LIN {X 0,Y 542.903,Z 219.007,A -85,B 0,C 180,E1 24562.487,E2 24562.487} C_VEL
LIN {X 0,Y 541.878,Z 217.291,A -85,B 0,C 180,E1 24561.084,E2 24561.084} C_VEL
LIN {X 0,Y 539.286,Z 215.915,A -85,B 0,C 180,E1 24558.559,E2 24558.559} C_VEL
LIN {X 0,Y 536.919,Z 213.82,A -85,B 0,C 180,E1 24556.541,E2 24556.541} C_VEL
LIN {X 0,Y 534.543,Z 210.096,A -85,B 0,C 180,E1 24554.71,E2 24554.71} C_VEL
LIN {X 0,Y 531.153,Z 208.109,A -85,B 0,C 180,E1 24552.586,E2 24552.586} C_VEL
LIN {X 0,Y 528.889,Z 205.137,A -85,B 0,C 180,E1 24551.198,E2 24551.198} C_VEL
LIN {X 0,Y 527.514,Z 203.01,A -85,B 0,C 180,E1 24550.4,E2 24550.4} C_VEL
LIN {X 0,Y 524.38,Z 201.255,A -85,B 0,C 180,E1 24548.817,E2 24548.817} C_VEL
LIN {X 0,Y 522.406,Z 198.666,A -85,B 0,C 180,E1 24547.792,E2 24547.792} C_VEL
LIN {X 0,Y 521.741,Z 196.733,A -85,B 0,C 180,E1 24547.193,E2 24547.193} C_VEL
LIN {X 0,Y 521.717,Z 196.18,A -85,B 0,C 180,E1 24546.271,E2 24546.271} C_VEL
LIN {X 0,Y 521.67,Z 196.188,A -85,B 0,C 180,E1 24542.863,E2 24542.863} C_VEL
LIN {X 0,Y 521.655,Z 196.188,A -85,B 0,C 180,E1 24539.478,E2 24539.478} C_VEL
LIN {X 0,Y 521.706,Z 196.182,A -85,B 0,C 180,E1 24536.239,E2 24536.239} C_VEL
LIN {X 0,Y 521.677,Z 196.188,A -85,B 0,C 180,E1 24532.867,E2 24532.867} C_VEL
LIN {X 0,Y 521.656,Z 196.187,A -85,B 0,C 180,E1 24529.549,E2 24529.549} C_VEL
LIN {X 0,Y 521.694,Z 196.184,A -85,B 0,C 180,E1 24526.227,E2 24526.227} C_VEL
LIN {X 0,Y 521.689,Z 196.187,A -85,B 0,C 180,E1 24522.876,E2 24522.876} C_VEL
LIN {X 0,Y 521.655,Z 196.188,A -85,B 0,C 180,E1 24519.607,E2 24519.607} C_VEL
LIN {X 0,Y 521.686,Z 196.144,A -85,B 0,C 180,E1 24516.317,E2 24516.317} C_VEL
LIN {X 0,Y 521.69,Z 196.17,A -85,B 0,C 180,E1 24512.926,E2 24512.926} C_VEL
LIN {X 0,Y 521.65,Z 196.155,A -85,B 0,C 180,E1 24509.639,E2 24509.639} C_VEL
LIN {X 0,Y 521.686,Z 196.134,A -85,B 0,C 180,E1 24506.402,E2 24506.402} C_VEL
LIN {X 0,Y 521.687,Z 196.186,A -85,B 0,C 180,E1 24503.094,E2 24503.094} C_VEL
LIN {X 0,Y 521.654,Z 196.185,A -85,B 0,C 180,E1 24499.779,E2 24499.779} C_VEL
LIN {X 0,Y 521.685,Z 196.169,A -85,B 0,C 180,E1 24496.479,E2 24496.479} C_VEL
LIN {X 0,Y 521.684,Z 196.173,A -85,B 0,C 180,E1 24493.213,E2 24493.213} C_VEL
LIN {X 0,Y 521.654,Z 196.185,A -85,B 0,C 180,E1 24489.822,E2 24489.822} C_VEL
LIN {X 0,Y 521.666,Z 196.176,A -85,B 0,C 180,E1 24486.383,E2 24486.383} C_VEL
LIN {X 0,Y 521.707,Z 196.167,A -85,B 0,C 180,E1 24483.076,E2 24483.076} C_VEL
LIN {X 0,Y 521.657,Z 196.185,A -85,B 0,C 180,E1 24479.78,E2 24479.78} C_VEL
LIN {X 0,Y 521.655,Z 196.174,A -85,B 0,C 180,E1 24476.263,E2 24476.263} C_VEL
LIN {X 0,Y 521.708,Z 196.163,A -85,B 0,C 180,E1 24472.954,E2 24472.954} C_VEL
LIN {X 0,Y 521.673,Z 196.183,A -85,B 0,C 180,E1 24469.62,E2 24469.62} C_VEL
LIN {X 0,Y 521.653,Z 196.179,A -85,B 0,C 180,E1 24466.25,E2 24466.25} C_VEL
LIN {X 0,Y 521.701,Z 196.166,A -85,B 0,C 180,E1 24462.989,E2 24462.989} C_VEL
LIN {X 0,Y 521.677,Z 196.186,A -85,B 0,C 180,E1 24459.701,E2 24459.701} C_VEL
LIN {X 0,Y 521.656,Z 196.185,A -85,B 0,C 180,E1 24456.36,E2 24456.36} C_VEL
LIN {X 0,Y 521.69,Z 196.137,A -85,B 0,C 180,E1 24453.013,E2 24453.013} C_VEL
LIN {X 0,Y 521.674,Z 196.16,A -85,B 0,C 180,E1 24449.804,E2 24449.804} C_VEL
LIN {X 0,Y 521.654,Z 196.173,A -85,B 0,C 180,E1 24446.479,E2 24446.479} C_VEL
LIN {X 0,Y 521.693,Z 196.178,A -85,B 0,C 180,E1 24443.137,E2 24443.137} C_VEL
LIN {X 0,Y 521.678,Z 196.156,A -85,B 0,C 180,E1 24439.876,E2 24439.876} C_VEL
LIN {X 0,Y 521.655,Z 196.17,A -85,B 0,C 180,E1 24436.518,E2 24436.518} C_VEL
LIN {X 0,Y 521.685,Z 196.174,A -85,B 0,C 180,E1 24433.169,E2 24433.169} C_VEL
LIN {X 0,Y 521.758,Z 196.445,A -85,B 0,C 180,E1 24431.589,E2 24431.589} C_VEL
LIN {X 0,Y 528.289,Z 215.738,A -85,B 0,C 180,E1 24428.585,E2 24428.585} C_VEL
LIN {X 0,Y 529.766,Z 220.377,A -85,B 0,C 180,E1 24427.913,E2 24427.913} C_VEL
LIN {X 0,Y 541.007,Z 241.596,A -85,B 0,C 180,E1 24426.622,E2 24426.622} C_VEL
LIN {X 0,Y 548.011,Z 256.158,A -85,B 0,C 180,E1 24425.852,E2 24425.852} C_VEL
LIN {X 0,Y 550.912,Z 271.289,A -85,B 0,C 180,E1 24425.399,E2 24425.399} C_VEL
LIN {X 0,Y 544.997,Z 522.592,A -85,B 0,C 180,E1 24421.909,E2 24421.909} C_VEL
LIN {X 0,Y 544.141,Z 540.067,A -85,B 0,C 180,E1 24421.568,E2 24421.568} C_VEL
LIN {X 0,Y 543,Z 557.267,A -85,B 0,C 180,E1 24421.118,E2 24421.118} C_VEL
LIN {X 0,Y 541.545,Z 575.435,A -85,B 0,C 180,E1 24420.509,E2 24420.509} C_VEL
LIN {X 0,Y 539.48,Z 597.06,A -85,B 0,C 180,E1 24419.595,E2 24419.595} C_VEL
LIN {X 0,Y 537.434,Z 615.482,A -85,B 0,C 180,E1 24418.621,E2 24418.621} C_VEL
LIN {X 0,Y 535.499,Z 631.43,A -85,B 0,C 180,E1 24417.63,E2 24417.63} C_VEL
LIN {X 0,Y 533.565,Z 646.552,A -85,B 0,C 180,E1 24416.544,E2 24416.544} C_VEL
LIN {X 0,Y 531.674,Z 660.645,A -85,B 0,C 180,E1 24415.387,E2 24415.387} C_VEL
LIN {X 0,Y 529.802,Z 674.285,A -85,B 0,C 180,E1 24414.113,E2 24414.113} C_VEL
LIN {X 0,Y 527.931,Z 687.897,A -85,B 0,C 180,E1 24412.667,E2 24412.667} C_VEL
LIN {X 0,Y 525.911,Z 703.024,A -85,B 0,C 180,E1 24410.823,E2 24410.823} C_VEL
LIN {X 0,Y 524.104,Z 716.894,A -85,B 0,C 180,E1 24408.807,E2 24408.807} C_VEL
LIN {X 0,Y 522.906,Z 726.951,A -85,B 0,C 180,E1 24407.124,E2 24407.124} C_VEL
LIN {X 0,Y 521.966,Z 735.746,A -85,B 0,C 180,E1 24405.44,E2 24405.44} C_VEL
LIN {X 0,Y 521.195,Z 743.869,A -85,B 0,C 180,E1 24403.647,E2 24403.647} C_VEL
LIN {X 0,Y 520.653,Z 750.809,A -85,B 0,C 180,E1 24401.856,E2 24401.856} C_VEL
LIN {X 0,Y 520.296,Z 756.648,A -85,B 0,C 180,E1 24400.07,E2 24400.07} C_VEL
LIN {X 0,Y 520.076,Z 761.724,A -85,B 0,C 180,E1 24398.178,E2 24398.178} C_VEL
LIN {X 0,Y 519.973,Z 765.693,A -85,B 0,C 180,E1 24396.292,E2 24396.292} C_VEL
LIN {X 0,Y 519.93,Z 768.746,A -85,B 0,C 180,E1 24394.301,E2 24394.301} C_VEL
LIN {X 0,Y 519.929,Z 770.992,A -85,B 0,C 180,E1 24391.873,E2 24391.873} C_VEL
LIN {X 0,Y 519.925,Z 771.359,A -85,B 0,C 180,E1 24389.449,E2 24389.449} C_VEL
LIN {X 0,Y 519.924,Z 770.471,A -85,B 0,C 180,E1 24387.465,E2 24387.465} C_VEL
LIN {X 0,Y 519.93,Z 768.599,A -85,B 0,C 180,E1 24385.589,E2 24385.589} C_VEL
LIN {X 0,Y 519.973,Z 765.693,A -85,B 0,C 180,E1 24383.708,E2 24383.708} C_VEL
LIN {X 0,Y 520.076,Z 761.724,A -85,B 0,C 180,E1 24381.822,E2 24381.822} C_VEL
LIN {X 0,Y 520.296,Z 756.648,A -85,B 0,C 180,E1 24379.93,E2 24379.93} C_VEL
LIN {X 0,Y 520.653,Z 750.809,A -85,B 0,C 180,E1 24378.144,E2 24378.144} C_VEL
LIN {X 0,Y 521.195,Z 743.869,A -85,B 0,C 180,E1 24376.353,E2 24376.353} C_VEL
LIN {X 0,Y 521.966,Z 735.746,A -85,B 0,C 180,E1 24374.56,E2 24374.56} C_VEL
LIN {X 0,Y 523.051,Z 725.713,A -85,B 0,C 180,E1 24372.652,E2 24372.652} C_VEL
LIN {X 0,Y 524.751,Z 711.758,A -85,B 0,C 180,E1 24370.408,E2 24370.408} C_VEL
LIN {X 0,Y 526.363,Z 699.468,A -85,B 0,C 180,E1 24368.729,E2 24368.729} C_VEL
LIN {X 0,Y 528.029,Z 687.155,A -85,B 0,C 180,E1 24367.25,E2 24367.25} C_VEL
LIN {X 0,Y 529.8,Z 674.285,A -85,B 0,C 180,E1 24365.887,E2 24365.887} C_VEL
LIN {X 0,Y 531.674,Z 660.644,A -85,B 0,C 180,E1 24364.613,E2 24364.613} C_VEL
LIN {X 0,Y 533.566,Z 646.552,A -85,B 0,C 180,E1 24363.456,E2 24363.456} C_VEL
LIN {X 0,Y 535.501,Z 631.421,A -85,B 0,C 180,E1 24362.369,E2 24362.369} C_VEL
LIN {X 0,Y 537.545,Z 614.561,A -85,B 0,C 180,E1 24361.325,E2 24361.325} C_VEL
LIN {X 0,Y 539.952,Z 592.29,A -85,B 0,C 180,E1 24360.187,E2 24360.187} C_VEL
LIN {X 0,Y 541.671,Z 573.948,A -85,B 0,C 180,E1 24359.437,E2 24359.437} C_VEL
LIN {X 0,Y 543.051,Z 556.564,A -85,B 0,C 180,E1 24358.861,E2 24358.861} C_VEL
LIN {X 0,Y 544.169,Z 539.567,A -85,B 0,C 180,E1 24358.42,E2 24358.42} C_VEL
LIN {X 0,Y 545.016,Z 522.077,A -85,B 0,C 180,E1 24358.083,E2 24358.083} C_VEL
LIN {X 0,Y 550.932,Z 270.389,A -85,B 0,C 180,E1 24354.589,E2 24354.589} C_VEL
LIN {X 0,Y 547.528,Z 254.684,A -85,B 0,C 180,E1 24354.088,E2 24354.088} C_VEL
LIN {X 0,Y 534.954,Z 230.044,A -85,B 0,C 180,E1 24352.707,E2 24352.707} C_VEL
LIN {X 0,Y 529.698,Z 220.207,A -85,B 0,C 180,E1 24352.071,E2 24352.071} C_VEL
LIN {X 0,Y 523.725,Z 202.248,A -85,B 0,C 180,E1 24349.345,E2 24349.345} C_VEL
LIN {X 0,Y 521.737,Z 196.322,A -85,B 0,C 180,E1 24348.368,E2 24348.368} C_VEL
LIN {X 0,Y 521.673,Z 196.166,A -85,B 0,C 180,E1 24344.995,E2 24344.995} C_VEL
LIN {X 0,Y 521.656,Z 196.184,A -85,B 0,C 180,E1 24341.631,E2 24341.631} C_VEL
LIN {X 0,Y 521.707,Z 196.174,A -85,B 0,C 180,E1 24338.387,E2 24338.387} C_VEL
LIN {X 0,Y 521.672,Z 196.151,A -85,B 0,C 180,E1 24335.083,E2 24335.083} C_VEL
LIN {X 0,Y 521.657,Z 196.186,A -85,B 0,C 180,E1 24331.681,E2 24331.681} C_VEL
LIN {X 0,Y 521.687,Z 196.121,A -85,B 0,C 180,E1 24328.381,E2 24328.381} C_VEL
LIN {X 0,Y 521.688,Z 196.177,A -85,B 0,C 180,E1 24325.061,E2 24325.061} C_VEL
LIN {X 0,Y 521.652,Z 196.17,A -85,B 0,C 180,E1 24321.83,E2 24321.83} C_VEL
LIN {X 0,Y 521.698,Z 196.168,A -85,B 0,C 180,E1 24318.552,E2 24318.552} C_VEL
LIN {X 0,Y 521.682,Z 196.182,A -85,B 0,C 180,E1 24315.224,E2 24315.224} C_VEL
LIN {X 0,Y 521.654,Z 196.177,A -85,B 0,C 180,E1 24311.947,E2 24311.947} C_VEL
LIN {X 0,Y 521.688,Z 196.164,A -85,B 0,C 180,E1 24308.598,E2 24308.598} C_VEL
LIN {X 0,Y 521.677,Z 196.185,A -85,B 0,C 180,E1 24305.389,E2 24305.389} C_VEL
LIN {X 0,Y 521.653,Z 196.177,A -85,B 0,C 180,E1 24301.977,E2 24301.977} C_VEL
LIN {X 0,Y 521.686,Z 196.168,A -85,B 0,C 180,E1 24298.682,E2 24298.682} C_VEL
LIN {X 0,Y 521.697,Z 196.184,A -85,B 0,C 180,E1 24295.273,E2 24295.273} C_VEL
LIN {X 0,Y 521.652,Z 196.175,A -85,B 0,C 180,E1 24292.067,E2 24292.067} C_VEL
LIN {X 0,Y 521.68,Z 196.171,A -85,B 0,C 180,E1 24288.726,E2 24288.726} C_VEL
LIN {X 0,Y 521.702,Z 196.184,A -85,B 0,C 180,E1 24285.345,E2 24285.345} C_VEL
LIN {X 0,Y 521.656,Z 196.178,A -85,B 0,C 180,E1 24282.025,E2 24282.025} C_VEL
LIN {X 0,Y 521.658,Z 196.17,A -85,B 0,C 180,E1 24278.525,E2 24278.525} C_VEL
LIN {X 0,Y 521.713,Z 196.173,A -85,B 0,C 180,E1 24275.274,E2 24275.274} C_VEL
LIN {X 0,Y 521.656,Z 196.121,A -85,B 0,C 180,E1 24271.991,E2 24271.991} C_VEL
LIN {X 0,Y 521.656,Z 196.188,A -85,B 0,C 180,E1 24268.522,E2 24268.522} C_VEL
LIN {X 0,Y 521.692,Z 196.131,A -85,B 0,C 180,E1 24265.169,E2 24265.169} C_VEL
LIN {X 0,Y 521.684,Z 196.185,A -85,B 0,C 180,E1 24261.788,E2 24261.788} C_VEL
LIN {X 0,Y 521.654,Z 196.188,A -85,B 0,C 180,E1 24258.455,E2 24258.455} C_VEL
LIN {X 0,Y 521.686,Z 196.187,A -85,B 0,C 180,E1 24255.144,E2 24255.144} C_VEL
LIN {X 0,Y 521.695,Z 196.184,A -85,B 0,C 180,E1 24251.792,E2 24251.792} C_VEL
LIN {X 0,Y 521.654,Z 196.19,A -85,B 0,C 180,E1 24248.526,E2 24248.526} C_VEL
LIN {X 0,Y 521.673,Z 196.185,A -85,B 0,C 180,E1 24245.095,E2 24245.095} C_VEL
LIN {X 0,Y 521.709,Z 196.182,A -85,B 0,C 180,E1 24241.802,E2 24241.802} C_VEL
LIN {X 0,Y 521.657,Z 196.19,A -85,B 0,C 180,E1 24238.503,E2 24238.503} C_VEL
LIN {X 0,Y 521.66,Z 196.188,A -85,B 0,C 180,E1 24234.957,E2 24234.957} C_VEL
LIN {X 0,Y 521.695,Z 196.443,A -85,B 0,C 180,E1 24233.013,E2 24233.013} C_VEL
LIN {X 0,Y 522.028,Z 197.78,A -85,B 0,C 180,E1 24232.432,E2 24232.432} C_VEL
LIN {X 0,Y 523.785,Z 200.654,A -85,B 0,C 180,E1 24231.498,E2 24231.498} C_VEL
LIN {X 0,Y 526.561,Z 202.591,A -85,B 0,C 180,E1 24230.1,E2 24230.1} C_VEL
LIN {X 0,Y 528.085,Z 203.612,A -85,B 0,C 180,E1 24229.29,E2 24229.29} C_VEL
LIN {X 0,Y 530.137,Z 207.055,A -85,B 0,C 180,E1 24228.016,E2 24228.016} C_VEL
LIN {X 0,Y 532.738,Z 209.204,A -85,B 0,C 180,E1 24226.444,E2 24226.444} C_VEL
LIN {X 0,Y 535.076,Z 210.611,A -85,B 0,C 180,E1 24224.942,E2 24224.942} C_VEL
LIN {X 0,Y 537.044,Z 213.985,A -85,B 0,C 180,E1 24223.346,E2 24223.346} C_VEL
LIN {X 0,Y 539.43,Z 216.007,A -85,B 0,C 180,E1 24221.316,E2 24221.316} C_VEL
LIN {X 0,Y 541.878,Z 217.29,A -85,B 0,C 180,E1 24218.916,E2 24218.916} C_VEL
LIN {X 0,Y 542.903,Z 219.006,A -85,B 0,C 180,E1 24217.513,E2 24217.513} C_VEL
LIN {X 0,Y 544.125,Z 220.957,A -85,B 0,C 180,E1 24215.483,E2 24215.483} C_VEL
LIN {X 0,Y 545.134,Z 222.019,A -85,B 0,C 180,E1 24212.943,E2 24212.943} C_VEL
LIN {X 0,Y 545.527,Z 222.319,A -85,B 0,C 180,E1 24210.525,E2 24210.525} C_VEL
LIN {X 0,Y 545.35,Z 222.132,A -85,B 0,C 180,E1 24208.004,E2 24208.004} C_VEL
LIN {X 0,Y 544.651,Z 221.519,A -85,B 0,C 180,E1 24205.684,E2 24205.684} C_VEL
LIN {X 0,Y 543.982,Z 220.78,A -85,B 0,C 180,E1 24204.293,E2 24204.293} C_VEL
LIN {X 0,Y 543.556,Z 221.288,A -85,B 0,C 180,E1 24203.742,E2 24203.742} C_VEL
LIN {X 0,Y 542.023,Z 225.814,A -85,B 0,C 180,E1 24202.381,E2 24202.381} C_VEL
LIN {X 0,Y 541.533,Z 226.008,A -85,B 0,C 180,E1 24201.833,E2 24201.833} C_VEL
LIN {X 0,Y 539.846,Z 224.583,A -85,B 0,C 180,E1 24199.975,E2 24199.975} C_VEL
LIN {X 0,Y 537.307,Z 223.183,A -85,B 0,C 180,E1 24197.685,E2 24197.685} C_VEL
LIN {X 0,Y 535.124,Z 220.823,A -85,B 0,C 180,E1 24195.944,E2 24195.944} C_VEL
LIN {X 0,Y 533.5,Z 218.054,A -85,B 0,C 180,E1 24194.679,E2 24194.679} C_VEL
LIN {X 0,Y 529.91,Z 215.891,A -85,B 0,C 180,E1 24192.43,E2 24192.43} C_VEL
LIN {X 0,Y 527.499,Z 212.743,A -85,B 0,C 180,E1 24190.975,E2 24190.975} C_VEL
LIN {X 0,Y 526.194,Z 210.803,A -85,B 0,C 180,E1 24190.233,E2 24190.233} C_VEL
LIN {X 0,Y 522.971,Z 208.929,A -85,B 0,C 180,E1 24188.61,E2 24188.61} C_VEL
LIN {X 0,Y 520.8,Z 206.047,A -85,B 0,C 180,E1 24187.503,E2 24187.503} C_VEL
LIN {X 0,Y 519.653,Z 204.128,A -85,B 0,C 180,E1 24186.889,E2 24186.889} C_VEL
LIN {X 0,Y 515.906,Z 201.753,A -85,B 0,C 180,E1 24185.255,E2 24185.255} C_VEL
LIN {X 0,Y 514.22,Z 199.009,A -85,B 0,C 180,E1 24184.454,E2 24184.454} C_VEL
LIN {X 0,Y 513.786,Z 197.461,A -85,B 0,C 180,E1 24183.911,E2 24183.911} C_VEL
LIN {X 0,Y 513.73,Z 197.176,A -85,B 0,C 180,E1 24180.888,E2 24180.888} C_VEL
LIN {X 0,Y 513.716,Z 197.178,A -85,B 0,C 180,E1 24177.436,E2 24177.436} C_VEL
LIN {X 0,Y 513.749,Z 197.174,A -85,B 0,C 180,E1 24174.062,E2 24174.062} C_VEL
LIN {X 0,Y 513.763,Z 197.171,A -85,B 0,C 180,E1 24170.626,E2 24170.626} C_VEL
LIN {X 0,Y 513.716,Z 197.178,A -85,B 0,C 180,E1 24167.37,E2 24167.37} C_VEL
LIN {X 0,Y 513.725,Z 197.178,A -85,B 0,C 180,E1 24163.86,E2 24163.86} C_VEL
LIN {X 0,Y 513.778,Z 197.172,A -85,B 0,C 180,E1 24160.462,E2 24160.462} C_VEL
LIN {X 0,Y 513.729,Z 197.154,A -85,B 0,C 180,E1 24157.111,E2 24157.111} C_VEL
LIN {X 0,Y 513.712,Z 197.142,A -85,B 0,C 180,E1 24153.692,E2 24153.692} C_VEL
LIN {X 0,Y 513.754,Z 197.159,A -85,B 0,C 180,E1 24150.399,E2 24150.399} C_VEL
LIN {X 0,Y 513.736,Z 197.108,A -85,B 0,C 180,E1 24147.093,E2 24147.093} C_VEL
LIN {X 0,Y 513.715,Z 197.176,A -85,B 0,C 180,E1 24143.76,E2 24143.76} C_VEL
LIN {X 0,Y 513.743,Z 197.167,A -85,B 0,C 180,E1 24140.389,E2 24140.389} C_VEL
LIN {X 0,Y 513.765,Z 197.153,A -85,B 0,C 180,E1 24136.974,E2 24136.974} C_VEL
LIN {X 0,Y 513.714,Z 197.172,A -85,B 0,C 180,E1 24133.737,E2 24133.737} C_VEL
LIN {X 0,Y 513.729,Z 197.173,A -85,B 0,C 180,E1 24130.315,E2 24130.315} C_VEL
LIN {X 0,Y 513.785,Z 197.15,A -85,B 0,C 180,E1 24126.93,E2 24126.93} C_VEL
LIN {X 0,Y 513.732,Z 197.168,A -85,B 0,C 180,E1 24123.459,E2 24123.459} C_VEL
LIN {X 0,Y 513.715,Z 197.174,A -85,B 0,C 180,E1 24120.111,E2 24120.111} C_VEL
LIN {X 0,Y 513.751,Z 197.153,A -85,B 0,C 180,E1 24116.764,E2 24116.764} C_VEL
LIN {X 0,Y 513.749,Z 197.163,A -85,B 0,C 180,E1 24113.406,E2 24113.406} C_VEL
LIN {X 0,Y 513.716,Z 197.172,A -85,B 0,C 180,E1 24110.024,E2 24110.024} C_VEL
LIN {X 0,Y 513.73,Z 197.16,A -85,B 0,C 180,E1 24106.608,E2 24106.608} C_VEL
LIN {X 0,Y 513.763,Z 197.16,A -85,B 0,C 180,E1 24103.376,E2 24103.376} C_VEL
LIN {X 0,Y 513.719,Z 197.175,A -85,B 0,C 180,E1 24100.046,E2 24100.046} C_VEL
LIN {X 0,Y 513.721,Z 197.174,A -85,B 0,C 180,E1 24096.484,E2 24096.484} C_VEL
LIN {X 0,Y 513.766,Z 197.126,A -85,B 0,C 180,E1 24093.159,E2 24093.159} C_VEL
LIN {X 0,Y 513.732,Z 197.144,A -85,B 0,C 180,E1 24089.857,E2 24089.857} C_VEL
LIN {X 0,Y 513.714,Z 197.159,A -85,B 0,C 180,E1 24086.442,E2 24086.442} C_VEL
LIN {X 0,Y 513.744,Z 197.17,A -85,B 0,C 180,E1 24083.029,E2 24083.029} C_VEL
LIN {X 0,Y 513.755,Z 197.142,A -85,B 0,C 180,E1 24079.713,E2 24079.713} C_VEL
LIN {X 0,Y 513.716,Z 197.156,A -85,B 0,C 180,E1 24076.382,E2 24076.382} C_VEL
LIN {X 0,Y 513.727,Z 197.16,A -85,B 0,C 180,E1 24072.932,E2 24072.932} C_VEL
LIN {X 0,Y 513.771,Z 197.484,A -85,B 0,C 180,E1 24072.206,E2 24072.206} C_VEL
LIN {X 0,Y 519.766,Z 214.932,A -85,B 0,C 180,E1 24069.401,E2 24069.401} C_VEL
LIN {X 0,Y 521.525,Z 220.084,A -85,B 0,C 180,E1 24068.622,E2 24068.622} C_VEL
LIN {X 0,Y 533.349,Z 242.254,A -85,B 0,C 180,E1 24067.222,E2 24067.222} C_VEL
LIN {X 0,Y 541.827,Z 259.36,A -85,B 0,C 180,E1 24066.272,E2 24066.272} C_VEL
LIN {X 0,Y 544.347,Z 272.898,A -85,B 0,C 180,E1 24065.863,E2 24065.863} C_VEL
LIN {X 0,Y 538.202,Z 522.519,A -85,B 0,C 180,E1 24062.358,E2 24062.358} C_VEL
LIN {X 0,Y 537.313,Z 540.039,A -85,B 0,C 180,E1 24062.013,E2 24062.013} C_VEL
LIN {X 0,Y 536.116,Z 557.349,A -85,B 0,C 180,E1 24061.555,E2 24061.555} C_VEL
LIN {X 0,Y 534.559,Z 576.003,A -85,B 0,C 180,E1 24060.92,E2 24060.92} C_VEL
LIN {X 0,Y 532.22,Z 599.008,A -85,B 0,C 180,E1 24059.916,E2 24059.916} C_VEL
LIN {X 0,Y 530.224,Z 616.226,A -85,B 0,C 180,E1 24058.985,E2 24058.985} C_VEL
LIN {X 0,Y 528.235,Z 631.906,A -85,B 0,C 180,E1 24057.994,E2 24057.994} C_VEL
LIN {X 0,Y 526.304,Z 646.375,A -85,B 0,C 180,E1 24056.939,E2 24056.939} C_VEL
LIN {X 0,Y 524.33,Z 660.467,A -85,B 0,C 180,E1 24055.768,E2 24055.768} C_VEL
LIN {X 0,Y 522.404,Z 673.859,A -85,B 0,C 180,E1 24054.504,E2 24054.504} C_VEL
LIN {X 0,Y 520.535,Z 686.719,A -85,B 0,C 180,E1 24053.127,E2 24053.127} C_VEL
LIN {X 0,Y 518.748,Z 699.289,A -85,B 0,C 180,E1 24051.599,E2 24051.599} C_VEL
LIN {X 0,Y 516.759,Z 713.908,A -85,B 0,C 180,E1 24049.554,E2 24049.554} C_VEL
LIN {X 0,Y 515.177,Z 726.153,A -85,B 0,C 180,E1 24047.505,E2 24047.505} C_VEL
LIN {X 0,Y 514.104,Z 735.568,A -85,B 0,C 180,E1 24045.682,E2 24045.682} C_VEL
LIN {X 0,Y 513.284,Z 743.691,A -85,B 0,C 180,E1 24043.861,E2 24043.861} C_VEL
LIN {X 0,Y 512.707,Z 750.631,A -85,B 0,C 180,E1 24042.043,E2 24042.043} C_VEL
LIN {X 0,Y 512.326,Z 756.471,A -85,B 0,C 180,E1 24040.229,E2 24040.229} C_VEL
LIN {X 0,Y 512.092,Z 761.548,A -85,B 0,C 180,E1 24038.307,E2 24038.307} C_VEL
LIN {X 0,Y 511.974,Z 765.517,A -85,B 0,C 180,E1 24036.391,E2 24036.391} C_VEL
LIN {X 0,Y 511.93,Z 768.571,A -85,B 0,C 180,E1 24034.368,E2 24034.368} C_VEL
LIN {X 0,Y 511.93,Z 770.817,A -85,B 0,C 180,E1 24031.903,E2 24031.903} C_VEL
LIN {X 0,Y 511.927,Z 771.184,A -85,B 0,C 180,E1 24029.441,E2 24029.441} C_VEL
LIN {X 0,Y 511.925,Z 770.296,A -85,B 0,C 180,E1 24027.426,E2 24027.426} C_VEL
LIN {X 0,Y 511.93,Z 768.423,A -85,B 0,C 180,E1 24025.52,E2 24025.52} C_VEL
LIN {X 0,Y 511.974,Z 765.517,A -85,B 0,C 180,E1 24023.609,E2 24023.609} C_VEL
LIN {X 0,Y 512.092,Z 761.547,A -85,B 0,C 180,E1 24021.693,E2 24021.693} C_VEL
LIN {X 0,Y 512.326,Z 756.471,A -85,B 0,C 180,E1 24019.771,E2 24019.771} C_VEL
LIN {X 0,Y 512.707,Z 750.631,A -85,B 0,C 180,E1 24017.957,E2 24017.957} C_VEL
LIN {X 0,Y 513.284,Z 743.691,A -85,B 0,C 180,E1 24016.139,E2 24016.139} C_VEL
LIN {X 0,Y 514.11,Z 735.522,A -85,B 0,C 180,E1 24014.308,E2 24014.308} C_VEL
LIN {X 0,Y 515.254,Z 725.534,A -85,B 0,C 180,E1 24012.381,E2 24012.381} C_VEL
LIN {X 0,Y 517.055,Z 711.579,A -85,B 0,C 180,E1 24010.105,E2 24010.105} C_VEL
LIN {X 0,Y 518.748,Z 699.289,A -85,B 0,C 180,E1 24008.401,E2 24008.401} C_VEL
LIN {X 0,Y 520.535,Z 686.719,A -85,B 0,C 180,E1 24006.873,E2 24006.873} C_VEL
LIN {X 0,Y 522.404,Z 673.85,A -85,B 0,C 180,E1 24005.495,E2 24005.495} C_VEL
LIN {X 0,Y 524.33,Z 660.466,A -85,B 0,C 180,E1 24004.232,E2 24004.232} C_VEL
LIN {X 0,Y 526.304,Z 646.374,A -85,B 0,C 180,E1 24003.061,E2 24003.061} C_VEL
LIN {X 0,Y 528.236,Z 631.906,A -85,B 0,C 180,E1 24002.007,E2 24002.007} C_VEL
LIN {X 0,Y 530.225,Z 616.226,A -85,B 0,C 180,E1 24001.015,E2 24001.015} C_VEL
LIN {X 0,Y 532.344,Z 597.945,A -85,B 0,C 180,E1 24000.03,E2 24000.03} C_VEL
LIN {X 0,Y 534.559,Z 576.002,A -85,B 0,C 180,E1 23999.08,E2 23999.08} C_VEL
LIN {X 0,Y 536.125,Z 557.233,A -85,B 0,C 180,E1 23998.442,E2 23998.442} C_VEL
LIN {X 0,Y 537.31,Z 540.038,A -85,B 0,C 180,E1 23997.987,E2 23997.987} C_VEL
LIN {X 0,Y 538.203,Z 522.518,A -85,B 0,C 180,E1 23997.642,E2 23997.642} C_VEL
LIN {X 0,Y 544.37,Z 271.981,A -85,B 0,C 180,E1 23994.124,E2 23994.124} C_VEL
LIN {X 0,Y 541.404,Z 258.24,A -85,B 0,C 180,E1 23993.677,E2 23993.677} C_VEL
LIN {X 0,Y 529.174,Z 234.261,A -85,B 0,C 180,E1 23992.302,E2 23992.302} C_VEL
LIN {X 0,Y 521.465,Z 219.944,A -85,B 0,C 180,E1 23991.364,E2 23991.364} C_VEL
LIN {X 0,Y 515.542,Z 202.582,A -85,B 0,C 180,E1 23988.641,E2 23988.641} C_VEL
LIN {X 0,Y 513.737,Z 197.284,A -85,B 0,C 180,E1 23987.732,E2 23987.732} C_VEL
LIN {X 0,Y 513.77,Z 197.145,A -85,B 0,C 180,E1 23984.426,E2 23984.426} C_VEL
LIN {X 0,Y 513.727,Z 197.157,A -85,B 0,C 180,E1 23981.138,E2 23981.138} C_VEL
LIN {X 0,Y 513.718,Z 197.178,A -85,B 0,C 180,E1 23977.674,E2 23977.674} C_VEL
LIN {X 0,Y 513.755,Z 197.139,A -85,B 0,C 180,E1 23974.362,E2 23974.362} C_VEL
LIN {X 0,Y 513.743,Z 197.165,A -85,B 0,C 180,E1 23971.049,E2 23971.049} C_VEL
LIN {X 0,Y 513.71,Z 197.116,A -85,B 0,C 180,E1 23967.688,E2 23967.688} C_VEL
LIN {X 0,Y 513.737,Z 197.174,A -85,B 0,C 180,E1 23964.247,E2 23964.247} C_VEL
LIN {X 0,Y 513.773,Z 197.16,A -85,B 0,C 180,E1 23960.864,E2 23960.864} C_VEL
LIN {X 0,Y 513.72,Z 197.154,A -85,B 0,C 180,E1 23957.524,E2 23957.524} C_VEL
LIN {X 0,Y 513.718,Z 197.165,A -85,B 0,C 180,E1 23954.081,E2 23954.081} C_VEL
LIN {X 0,Y 513.769,Z 197.17,A -85,B 0,C 180,E1 23950.768,E2 23950.768} C_VEL
LIN {X 0,Y 513.733,Z 197.154,A -85,B 0,C 180,E1 23947.381,E2 23947.381} C_VEL
LIN {X 0,Y 513.715,Z 197.167,A -85,B 0,C 180,E1 23944.018,E2 23944.018} C_VEL
LIN {X 0,Y 513.75,Z 197.175,A -85,B 0,C 180,E1 23940.669,E2 23940.669} C_VEL
LIN {X 0,Y 513.748,Z 197.153,A -85,B 0,C 180,E1 23937.323,E2 23937.323} C_VEL
LIN {X 0,Y 513.714,Z 197.17,A -85,B 0,C 180,E1 23933.967,E2 23933.967} C_VEL
LIN {X 0,Y 513.734,Z 197.175,A -85,B 0,C 180,E1 23930.59,E2 23930.59} C_VEL
LIN {X 0,Y 513.775,Z 197.154,A -85,B 0,C 180,E1 23927.134,E2 23927.134} C_VEL
LIN {X 0,Y 513.722,Z 197.166,A -85,B 0,C 180,E1 23923.839,E2 23923.839} C_VEL
LIN {X 0,Y 513.717,Z 197.174,A -85,B 0,C 180,E1 23920.376,E2 23920.376} C_VEL
LIN {X 0,Y 513.757,Z 197.171,A -85,B 0,C 180,E1 23916.991,E2 23916.991} C_VEL
LIN {X 0,Y 513.741,Z 197.124,A -85,B 0,C 180,E1 23913.656,E2 23913.656} C_VEL
LIN {X 0,Y 513.712,Z 197.142,A -85,B 0,C 180,E1 23910.371,E2 23910.371} C_VEL
LIN {X 0,Y 513.755,Z 197.158,A -85,B 0,C 180,E1 23907.112,E2 23907.112} C_VEL
LIN {X 0,Y 513.748,Z 197.131,A -85,B 0,C 180,E1 23903.672,E2 23903.672} C_VEL
LIN {X 0,Y 513.716,Z 197.177,A -85,B 0,C 180,E1 23900.413,E2 23900.413} C_VEL
LIN {X 0,Y 513.739,Z 197.176,A -85,B 0,C 180,E1 23897.03,E2 23897.03} C_VEL
LIN {X 0,Y 513.769,Z 197.171,A -85,B 0,C 180,E1 23893.616,E2 23893.616} C_VEL
LIN {X 0,Y 513.721,Z 197.177,A -85,B 0,C 180,E1 23890.272,E2 23890.272} C_VEL
LIN {X 0,Y 513.721,Z 197.177,A -85,B 0,C 180,E1 23886.827,E2 23886.827} C_VEL
LIN {X 0,Y 513.761,Z 197.171,A -85,B 0,C 180,E1 23883.415,E2 23883.415} C_VEL
LIN {X 0,Y 513.735,Z 197.177,A -85,B 0,C 180,E1 23880.138,E2 23880.138} C_VEL
LIN {X 0,Y 513.717,Z 197.176,A -85,B 0,C 180,E1 23876.715,E2 23876.715} C_VEL
LIN {X 0,Y 513.834,Z 197.665,A -85,B 0,C 180,E1 23875.962,E2 23875.962} C_VEL
LIN {X 0,Y 514.412,Z 199.498,A -85,B 0,C 180,E1 23875.437,E2 23875.437} C_VEL
LIN {X 0,Y 516.401,Z 202.221,A -85,B 0,C 180,E1 23874.536,E2 23874.536} C_VEL
LIN {X 0,Y 520.183,Z 204.718,A -85,B 0,C 180,E1 23872.844,E2 23872.844} C_VEL
LIN {X 0,Y 522.224,Z 208.142,A -85,B 0,C 180,E1 23871.779,E2 23871.779} C_VEL
LIN {X 0,Y 525.25,Z 210.41,A -85,B 0,C 180,E1 23870.268,E2 23870.268} C_VEL
LIN {X 0,Y 526.77,Z 211.401,A -85,B 0,C 180,E1 23869.45,E2 23869.45} C_VEL
LIN {X 0,Y 528.855,Z 214.814,A -85,B 0,C 180,E1 23868.175,E2 23868.175} C_VEL
LIN {X 0,Y 531.448,Z 217.007,A -85,B 0,C 180,E1 23866.615,E2 23866.615} C_VEL
LIN {X 0,Y 533.851,Z 218.402,A -85,B 0,C 180,E1 23865.088,E2 23865.088} C_VEL
LIN {X 0,Y 535.894,Z 221.797,A -85,B 0,C 180,E1 23863.485,E2 23863.485} C_VEL
LIN {X 0,Y 538.277,Z 223.854,A -85,B 0,C 180,E1 23861.463,E2 23861.463} C_VEL
LIN {X 0,Y 540.884,Z 225.237,A -85,B 0,C 180,E1 23858.932,E2 23858.932} C_VEL
LIN {X 0,Y 541.906,Z 227.015,A -85,B 0,C 180,E1 23857.527,E2 23857.527} C_VEL
LIN {X 0,Y 543.256,Z 229.018,A -85,B 0,C 180,E1 23855.28,E2 23855.28} C_VEL
LIN {X 0,Y 544.265,Z 230.034,A -85,B 0,C 180,E1 23852.632,E2 23852.632} C_VEL
LIN {X 0,Y 544.621,Z 230.261,A -85,B 0,C 180,E1 23850,E2 23850} C_VEL
LIN {X 0,Y 544.266,Z 230.035,A -85,B 0,C 180,E1 23847.368,E2 23847.368} C_VEL
LIN {X 0,Y 543.253,Z 229.015,A -85,B 0,C 180,E1 23844.715,E2 23844.715} C_VEL
LIN {X 0,Y 541.907,Z 227.015,A -85,B 0,C 180,E1 23842.473,E2 23842.473} C_VEL
LIN {X 0,Y 541.533,Z 226.008,A -85,B 0,C 180,E1 23841.833,E2 23841.833} C_VEL
LIN {X 0,Y 540.898,Z 225.849,A -85,B 0,C 180,E1 23841.136,E2 23841.136} C_VEL
LIN {X 0,Y 539.568,Z 228.026,A -85,B 0,C 180,E1 23840.105,E2 23840.105} C_VEL
LIN {X 0,Y 537.766,Z 231.174,A -85,B 0,C 180,E1 23838.841,E2 23838.841} C_VEL
LIN {X 0,Y 536.851,Z 231.496,A -85,B 0,C 180,E1 23838.133,E2 23838.133} C_VEL
LIN {X 0,Y 534.386,Z 229.242,A -85,B 0,C 180,E1 23836.145,E2 23836.145} C_VEL
LIN {X 0,Y 532.262,Z 225.834,A -85,B 0,C 180,E1 23834.517,E2 23834.517} C_VEL
LIN {X 0,Y 528.794,Z 223.801,A -85,B 0,C 180,E1 23832.366,E2 23832.366} C_VEL
LIN {X 0,Y 526.264,Z 220.679,A -85,B 0,C 180,E1 23830.865,E2 23830.865} C_VEL
LIN {X 0,Y 525.078,Z 218.705,A -85,B 0,C 180,E1 23830.172,E2 23830.172} C_VEL
LIN {X 0,Y 521.816,Z 216.835,A -85,B 0,C 180,E1 23828.535,E2 23828.535} C_VEL
LIN {X 0,Y 519.419,Z 213.844,A -85,B 0,C 180,E1 23827.33,E2 23827.33} C_VEL
LIN {X 0,Y 518.199,Z 211.825,A -85,B 0,C 180,E1 23826.703,E2 23826.703} C_VEL
LIN {X 0,Y 514.614,Z 209.617,A -85,B 0,C 180,E1 23825.146,E2 23825.146} C_VEL
LIN {X 0,Y 512.648,Z 206.674,A -85,B 0,C 180,E1 23824.222,E2 23824.222} C_VEL
LIN {X 0,Y 511.498,Z 204.958,A -85,B 0,C 180,E1 23823.723,E2 23823.723} C_VEL
LIN {X 0,Y 508.348,Z 203.056,A -85,B 0,C 180,E1 23822.473,E2 23822.473} C_VEL
LIN {X 0,Y 506.319,Z 200.212,A -85,B 0,C 180,E1 23821.616,E2 23821.616} C_VEL
LIN {X 0,Y 505.832,Z 198.522,A -85,B 0,C 180,E1 23821.127,E2 23821.127} C_VEL
LIN {X 0,Y 505.777,Z 198.166,A -85,B 0,C 180,E1 23819.469,E2 23819.469} C_VEL
LIN {X 0,Y 505.816,Z 198.161,A -85,B 0,C 180,E1 23816.125,E2 23816.125} C_VEL
LIN {X 0,Y 505.823,Z 198.162,A -85,B 0,C 180,E1 23812.623,E2 23812.623} C_VEL
LIN {X 0,Y 505.78,Z 198.164,A -85,B 0,C 180,E1 23809.285,E2 23809.285} C_VEL
LIN {X 0,Y 505.78,Z 198.167,A -85,B 0,C 180,E1 23805.697,E2 23805.697} C_VEL
LIN {X 0,Y 505.824,Z 198.163,A -85,B 0,C 180,E1 23802.336,E2 23802.336} C_VEL
LIN {X 0,Y 505.807,Z 198.165,A -85,B 0,C 180,E1 23798.949,E2 23798.949} C_VEL
LIN {X 0,Y 505.768,Z 198.111,A -85,B 0,C 180,E1 23795.537,E2 23795.537} C_VEL
LIN {X 0,Y 505.794,Z 198.166,A -85,B 0,C 180,E1 23792.126,E2 23792.126} C_VEL
LIN {X 0,Y 505.825,Z 198.098,A -85,B 0,C 180,E1 23788.838,E2 23788.838} C_VEL
LIN {X 0,Y 505.784,Z 198.146,A -85,B 0,C 180,E1 23785.402,E2 23785.402} C_VEL
LIN {X 0,Y 505.777,Z 198.149,A -85,B 0,C 180,E1 23781.94,E2 23781.94} C_VEL
LIN {X 0,Y 505.819,Z 198.155,A -85,B 0,C 180,E1 23778.558,E2 23778.558} C_VEL
LIN {X 0,Y 505.813,Z 198.157,A -85,B 0,C 180,E1 23775.126,E2 23775.126} C_VEL
LIN {X 0,Y 505.776,Z 198.145,A -85,B 0,C 180,E1 23771.749,E2 23771.749} C_VEL
LIN {X 0,Y 505.785,Z 198.151,A -85,B 0,C 180,E1 23768.298,E2 23768.298} C_VEL
LIN {X 0,Y 505.834,Z 198.16,A -85,B 0,C 180,E1 23764.99,E2 23764.99} C_VEL
LIN {X 0,Y 505.786,Z 198.144,A -85,B 0,C 180,E1 23761.586,E2 23761.586} C_VEL
LIN {X 0,Y 505.778,Z 198.154,A -85,B 0,C 180,E1 23758.187,E2 23758.187} C_VEL
LIN {X 0,Y 505.814,Z 198.161,A -85,B 0,C 180,E1 23754.783,E2 23754.783} C_VEL
LIN {X 0,Y 505.802,Z 198.139,A -85,B 0,C 180,E1 23751.474,E2 23751.474} C_VEL
LIN {X 0,Y 505.776,Z 198.154,A -85,B 0,C 180,E1 23748.084,E2 23748.084} C_VEL
LIN {X 0,Y 505.793,Z 198.163,A -85,B 0,C 180,E1 23744.639,E2 23744.639} C_VEL
LIN {X 0,Y 505.835,Z 198.15,A -85,B 0,C 180,E1 23741.204,E2 23741.204} C_VEL
LIN {X 0,Y 505.79,Z 198.146,A -85,B 0,C 180,E1 23737.816,E2 23737.816} C_VEL
LIN {X 0,Y 505.778,Z 198.152,A -85,B 0,C 180,E1 23734.337,E2 23734.337} C_VEL
LIN {X 0,Y 505.795,Z 198.103,A -85,B 0,C 180,E1 23730.901,E2 23730.901} C_VEL
LIN {X 0,Y 505.822,Z 198.162,A -85,B 0,C 180,E1 23727.608,E2 23727.608} C_VEL
LIN {X 0,Y 505.779,Z 198.136,A -85,B 0,C 180,E1 23724.185,E2 23724.185} C_VEL
LIN {X 0,Y 505.784,Z 198.139,A -85,B 0,C 180,E1 23720.757,E2 23720.757} C_VEL
LIN {X 0,Y 505.836,Z 198.158,A -85,B 0,C 180,E1 23717.465,E2 23717.465} C_VEL
LIN {X 0,Y 505.801,Z 198.165,A -85,B 0,C 180,E1 23713.98,E2 23713.98} C_VEL
LIN {X 0,Y 505.825,Z 198.437,A -85,B 0,C 180,E1 23712.859,E2 23712.859} C_VEL
LIN {X 0,Y 511.88,Z 215.77,A -85,B 0,C 180,E1 23709.984,E2 23709.984} C_VEL
LIN {X 0,Y 513.35,Z 220.23,A -85,B 0,C 180,E1 23709.329,E2 23709.329} C_VEL
LIN {X 0,Y 525.497,Z 242.355,A -85,B 0,C 180,E1 23707.87,E2 23707.87} C_VEL
LIN {X 0,Y 535.696,Z 262.659,A -85,B 0,C 180,E1 23706.698,E2 23706.698} C_VEL
LIN {X 0,Y 537.823,Z 274.377,A -85,B 0,C 180,E1 23706.34,E2 23706.34} C_VEL
LIN {X 0,Y 531.434,Z 522.652,A -85,B 0,C 180,E1 23702.816,E2 23702.816} C_VEL
LIN {X 0,Y 530.499,Z 540.306,A -85,B 0,C 180,E1 23702.462,E2 23702.462} C_VEL
LIN {X 0,Y 529.211,Z 558.128,A -85,B 0,C 180,E1 23701.982,E2 23701.982} C_VEL
LIN {X 0,Y 527.303,Z 579.876,A -85,B 0,C 180,E1 23701.217,E2 23701.217} C_VEL
LIN {X 0,Y 525.031,Z 600.512,A -85,B 0,C 180,E1 23700.268,E2 23700.268} C_VEL
LIN {X 0,Y 523.037,Z 616.971,A -85,B 0,C 180,E1 23699.359,E2 23699.359} C_VEL
LIN {X 0,Y 520.996,Z 632.364,A -85,B 0,C 180,E1 23698.368,E2 23698.368} C_VEL
LIN {X 0,Y 518.966,Z 646.908,A -85,B 0,C 180,E1 23697.29,E2 23697.29} C_VEL
LIN {X 0,Y 516.913,Z 660.919,A -85,B 0,C 180,E1 23696.104,E2 23696.104} C_VEL
LIN {X 0,Y 514.87,Z 674.489,A -85,B 0,C 180,E1 23694.798,E2 23694.798} C_VEL
LIN {X 0,Y 512.807,Z 688.071,A -85,B 0,C 180,E1 23693.31,E2 23693.31} C_VEL
LIN {X 0,Y 510.533,Z 703.483,A -85,B 0,C 180,E1 23691.36,E2 23691.36} C_VEL
LIN {X 0,Y 508.645,Z 716.536,A -85,B 0,C 180,E1 23689.401,E2 23689.401} C_VEL
LIN {X 0,Y 507.306,Z 726.594,A -85,B 0,C 180,E1 23687.667,E2 23687.667} C_VEL
LIN {X 0,Y 506.208,Z 735.749,A -85,B 0,C 180,E1 23685.855,E2 23685.855} C_VEL
LIN {X 0,Y 505.379,Z 743.513,A -85,B 0,C 180,E1 23684.083,E2 23684.083} C_VEL
LIN {X 0,Y 504.766,Z 750.454,A -85,B 0,C 180,E1 23682.235,E2 23682.235} C_VEL
LIN {X 0,Y 504.359,Z 756.294,A -85,B 0,C 180,E1 23680.392,E2 23680.392} C_VEL
LIN {X 0,Y 504.103,Z 761.371,A -85,B 0,C 180,E1 23678.439,E2 23678.439} C_VEL
LIN {X 0,Y 503.975,Z 765.341,A -85,B 0,C 180,E1 23676.492,E2 23676.492} C_VEL
LIN {X 0,Y 503.93,Z 768.396,A -85,B 0,C 180,E1 23674.438,E2 23674.438} C_VEL
LIN {X 0,Y 503.932,Z 770.642,A -85,B 0,C 180,E1 23671.933,E2 23671.933} C_VEL
LIN {X 0,Y 503.929,Z 771.009,A -85,B 0,C 180,E1 23669.432,E2 23669.432} C_VEL
LIN {X 0,Y 503.925,Z 770.121,A -85,B 0,C 180,E1 23667.385,E2 23667.385} C_VEL
LIN {X 0,Y 503.929,Z 768.248,A -85,B 0,C 180,E1 23665.448,E2 23665.448} C_VEL
LIN {X 0,Y 503.975,Z 765.341,A -85,B 0,C 180,E1 23663.508,E2 23663.508} C_VEL
LIN {X 0,Y 504.104,Z 761.371,A -85,B 0,C 180,E1 23661.561,E2 23661.561} C_VEL
LIN {X 0,Y 504.359,Z 756.294,A -85,B 0,C 180,E1 23659.608,E2 23659.608} C_VEL
LIN {X 0,Y 504.766,Z 750.454,A -85,B 0,C 180,E1 23657.765,E2 23657.765} C_VEL
LIN {X 0,Y 505.379,Z 743.513,A -85,B 0,C 180,E1 23655.917,E2 23655.917} C_VEL
LIN {X 0,Y 506.249,Z 735.389,A -85,B 0,C 180,E1 23654.068,E2 23654.068} C_VEL
LIN {X 0,Y 507.468,Z 725.356,A -85,B 0,C 180,E1 23652.101,E2 23652.101} C_VEL
LIN {X 0,Y 509.402,Z 711.191,A -85,B 0,C 180,E1 23649.761,E2 23649.761} C_VEL
LIN {X 0,Y 511.241,Z 698.47,A -85,B 0,C 180,E1 23647.981,E2 23647.981} C_VEL
LIN {X 0,Y 513.107,Z 686.041,A -85,B 0,C 180,E1 23646.458,E2 23646.458} C_VEL
LIN {X 0,Y 515.041,Z 673.367,A -85,B 0,C 180,E1 23645.088,E2 23645.088} C_VEL
LIN {X 0,Y 517.069,Z 659.871,A -85,B 0,C 180,E1 23643.802,E2 23643.802} C_VEL
LIN {X 0,Y 519.17,Z 645.485,A -85,B 0,C 180,E1 23642.598,E2 23642.598} C_VEL
LIN {X 0,Y 521.414,Z 629.31,A -85,B 0,C 180,E1 23641.42,E2 23641.42} C_VEL
LIN {X 0,Y 524.194,Z 607.819,A -85,B 0,C 180,E1 23640.112,E2 23640.112} C_VEL
LIN {X 0,Y 526.28,Z 589.369,A -85,B 0,C 180,E1 23639.199,E2 23639.199} C_VEL
LIN {X 0,Y 527.934,Z 572.852,A -85,B 0,C 180,E1 23638.521,E2 23638.521} C_VEL
LIN {X 0,Y 529.39,Z 555.798,A -85,B 0,C 180,E1 23637.949,E2 23637.949} C_VEL
LIN {X 0,Y 530.589,Z 538.83,A -85,B 0,C 180,E1 23637.504,E2 23637.504} C_VEL
LIN {X 0,Y 531.491,Z 521.213,A -85,B 0,C 180,E1 23637.16,E2 23637.16} C_VEL
LIN {X 0,Y 537.838,Z 273.355,A -85,B 0,C 180,E1 23633.644,E2 23633.644} C_VEL
LIN {X 0,Y 535.305,Z 261.826,A -85,B 0,C 180,E1 23633.257,E2 23633.257} C_VEL
LIN {X 0,Y 523.51,Z 238.598,A -85,B 0,C 180,E1 23631.898,E2 23631.898} C_VEL
LIN {X 0,Y 513.281,Z 220.084,A -85,B 0,C 180,E1 23630.658,E2 23630.658} C_VEL
LIN {X 0,Y 507.812,Z 204.017,A -85,B 0,C 180,E1 23628.098,E2 23628.098} C_VEL
LIN {X 0,Y 505.802,Z 198.257,A -85,B 0,C 180,E1 23627.084,E2 23627.084} C_VEL
LIN {X 0,Y 505.778,Z 198.143,A -85,B 0,C 180,E1 23623.627,E2 23623.627} C_VEL
LIN {X 0,Y 505.812,Z 198.13,A -85,B 0,C 180,E1 23620.272,E2 23620.272} C_VEL
LIN {X 0,Y 505.809,Z 198.157,A -85,B 0,C 180,E1 23616.938,E2 23616.938} C_VEL
LIN {X 0,Y 505.775,Z 198.145,A -85,B 0,C 180,E1 23613.611,E2 23613.611} C_VEL
LIN {X 0,Y 505.802,Z 198.134,A -85,B 0,C 180,E1 23610.259,E2 23610.259} C_VEL
LIN {X 0,Y 505.819,Z 198.111,A -85,B 0,C 180,E1 23606.916,E2 23606.916} C_VEL
LIN {X 0,Y 505.782,Z 198.163,A -85,B 0,C 180,E1 23603.537,E2 23603.537} C_VEL
LIN {X 0,Y 505.781,Z 198.162,A -85,B 0,C 180,E1 23599.999,E2 23599.999} C_VEL
LIN {X 0,Y 505.827,Z 198.145,A -85,B 0,C 180,E1 23596.656,E2 23596.656} C_VEL
LIN {X 0,Y 505.792,Z 198.145,A -85,B 0,C 180,E1 23593.373,E2 23593.373} C_VEL
LIN {X 0,Y 505.776,Z 198.161,A -85,B 0,C 180,E1 23589.904,E2 23589.904} C_VEL
LIN {X 0,Y 505.797,Z 198.159,A -85,B 0,C 180,E1 23586.47,E2 23586.47} C_VEL
LIN {X 0,Y 505.826,Z 198.14,A -85,B 0,C 180,E1 23583.06,E2 23583.06} C_VEL
LIN {X 0,Y 505.78,Z 198.164,A -85,B 0,C 180,E1 23579.774,E2 23579.774} C_VEL
LIN {X 0,Y 505.779,Z 198.162,A -85,B 0,C 180,E1 23576.259,E2 23576.259} C_VEL
LIN {X 0,Y 505.818,Z 198.141,A -85,B 0,C 180,E1 23572.842,E2 23572.842} C_VEL
LIN {X 0,Y 505.813,Z 198.159,A -85,B 0,C 180,E1 23569.406,E2 23569.406} C_VEL
LIN {X 0,Y 505.776,Z 198.162,A -85,B 0,C 180,E1 23566.043,E2 23566.043} C_VEL
LIN {X 0,Y 505.791,Z 198.148,A -85,B 0,C 180,E1 23562.632,E2 23562.632} C_VEL
LIN {X 0,Y 505.837,Z 198.145,A -85,B 0,C 180,E1 23559.204,E2 23559.204} C_VEL
LIN {X 0,Y 505.79,Z 198.165,A -85,B 0,C 180,E1 23555.844,E2 23555.844} C_VEL
LIN {X 0,Y 505.77,Z 198.096,A -85,B 0,C 180,E1 23552.444,E2 23552.444} C_VEL
LIN {X 0,Y 505.816,Z 198.158,A -85,B 0,C 180,E1 23549.071,E2 23549.071} C_VEL
LIN {X 0,Y 505.803,Z 198.112,A -85,B 0,C 180,E1 23545.709,E2 23545.709} C_VEL
LIN {X 0,Y 505.777,Z 198.162,A -85,B 0,C 180,E1 23542.347,E2 23542.347} C_VEL
LIN {X 0,Y 505.798,Z 198.165,A -85,B 0,C 180,E1 23538.98,E2 23538.98} C_VEL
LIN {X 0,Y 505.833,Z 198.162,A -85,B 0,C 180,E1 23535.52,E2 23535.52} C_VEL
LIN {X 0,Y 505.792,Z 198.163,A -85,B 0,C 180,E1 23532.072,E2 23532.072} C_VEL
LIN {X 0,Y 505.777,Z 198.168,A -85,B 0,C 180,E1 23528.655,E2 23528.655} C_VEL
LIN {X 0,Y 505.808,Z 198.162,A -85,B 0,C 180,E1 23525.25,E2 23525.25} C_VEL
LIN {X 0,Y 505.824,Z 198.16,A -85,B 0,C 180,E1 23521.852,E2 23521.852} C_VEL
LIN {X 0,Y 505.812,Z 198.367,A -85,B 0,C 180,E1 23518.963,E2 23518.963} C_VEL
LIN {X 0,Y 506.205,Z 199.92,A -85,B 0,C 180,E1 23518.445,E2 23518.445} C_VEL
LIN {X 0,Y 508.009,Z 202.709,A -85,B 0,C 180,E1 23517.66,E2 23517.66} C_VEL
LIN {X 0,Y 510.566,Z 204.536,A -85,B 0,C 180,E1 23516.642,E2 23516.642} C_VEL
LIN {X 0,Y 512.196,Z 205.709,A -85,B 0,C 180,E1 23515.989,E2 23515.989} C_VEL
LIN {X 0,Y 514.091,Z 209.05,A -85,B 0,C 180,E1 23515.084,E2 23515.084} C_VEL
LIN {X 0,Y 516.626,Z 211.051,A -85,B 0,C 180,E1 23513.978,E2 23513.978} C_VEL
LIN {X 0,Y 518.727,Z 212.357,A -85,B 0,C 180,E1 23513.062,E2 23513.062} C_VEL
LIN {X 0,Y 520.782,Z 215.81,A -85,B 0,C 180,E1 23511.974,E2 23511.974} C_VEL
LIN {X 0,Y 523.903,Z 218.221,A -85,B 0,C 180,E1 23510.43,E2 23510.43} C_VEL
LIN {X 0,Y 525.448,Z 219.16,A -85,B 0,C 180,E1 23509.618,E2 23509.618} C_VEL
LIN {X 0,Y 527.477,Z 222.449,A -85,B 0,C 180,E1 23508.396,E2 23508.396} C_VEL
LIN {X 0,Y 529.995,Z 224.704,A -85,B 0,C 180,E1 23506.888,E2 23506.888} C_VEL
LIN {X 0,Y 532.707,Z 226.288,A -85,B 0,C 180,E1 23505.183,E2 23505.183} C_VEL
LIN {X 0,Y 534.702,Z 229.601,A -85,B 0,C 180,E1 23503.626,E2 23503.626} C_VEL
LIN {X 0,Y 537.143,Z 231.709,A -85,B 0,C 180,E1 23501.596,E2 23501.596} C_VEL
LIN {X 0,Y 539.802,Z 233.103,A -85,B 0,C 180,E1 23499.058,E2 23499.058} C_VEL
LIN {X 0,Y 540.847,Z 234.861,A -85,B 0,C 180,E1 23497.648,E2 23497.648} C_VEL
LIN {X 0,Y 542.225,Z 236.908,A -85,B 0,C 180,E1 23495.396,E2 23495.396} C_VEL
LIN {X 0,Y 543.259,Z 237.961,A -85,B 0,C 180,E1 23492.743,E2 23492.743} C_VEL
LIN {X 0,Y 543.615,Z 238.203,A -85,B 0,C 180,E1 23490.211,E2 23490.211} C_VEL
LIN {X 0,Y 543.356,Z 237.99,A -85,B 0,C 180,E1 23487.765,E2 23487.765} C_VEL
LIN {X 0,Y 542.486,Z 237.215,A -85,B 0,C 180,E1 23485.243,E2 23485.243} C_VEL
LIN {X 0,Y 541.16,Z 235.495,A -85,B 0,C 180,E1 23482.843,E2 23482.843} C_VEL
LIN {X 0,Y 539.89,Z 233.187,A -85,B 0,C 180,E1 23481.051,E2 23481.051} C_VEL
LIN {X 0,Y 537.267,Z 231.792,A -85,B 0,C 180,E1 23478.515,E2 23478.515} C_VEL
LIN {X 0,Y 536.851,Z 231.496,A -85,B 0,C 180,E1 23478.133,E2 23478.133} C_VEL
LIN {X 0,Y 536.094,Z 232.037,A -85,B 0,C 180,E1 23477.576,E2 23477.576} C_VEL
LIN {X 0,Y 533.594,Z 236.392,A -85,B 0,C 180,E1 23476.204,E2 23476.204} C_VEL
LIN {X 0,Y 532.853,Z 236.551,A -85,B 0,C 180,E1 23475.732,E2 23475.732} C_VEL
LIN {X 0,Y 532.754,Z 236.42,A -85,B 0,C 180,E1 23475.654,E2 23475.654} C_VEL
LIN {X 0,Y 531.07,Z 233.655,A -85,B 0,C 180,E1 23474.383,E2 23474.383} C_VEL
LIN {X 0,Y 527.772,Z 231.787,A -85,B 0,C 180,E1 23472.357,E2 23472.357} C_VEL
LIN {X 0,Y 525.056,Z 228.628,A -85,B 0,C 180,E1 23470.767,E2 23470.767} C_VEL
LIN {X 0,Y 523.797,Z 226.536,A -85,B 0,C 180,E1 23470.023,E2 23470.023} C_VEL
LIN {X 0,Y 520.468,Z 224.565,A -85,B 0,C 180,E1 23468.358,E2 23468.358} C_VEL
LIN {X 0,Y 517.886,Z 221.325,A -85,B 0,C 180,E1 23467.066,E2 23467.066} C_VEL
LIN {X 0,Y 516.737,Z 219.57,A -85,B 0,C 180,E1 23466.512,E2 23466.512} C_VEL
LIN {X 0,Y 513.228,Z 217.381,A -85,B 0,C 180,E1 23464.994,E2 23464.994} C_VEL
LIN {X 0,Y 511.004,Z 214.251,A -85,B 0,C 180,E1 23463.977,E2 23463.977} C_VEL
LIN {X 0,Y 510.121,Z 212.748,A -85,B 0,C 180,E1 23463.584,E2 23463.584} C_VEL
LIN {X 0,Y 506.932,Z 210.837,A -85,B 0,C 180,E1 23462.329,E2 23462.329} C_VEL
LIN {X 0,Y 504.603,Z 207.724,A -85,B 0,C 180,E1 23461.349,E2 23461.349} C_VEL
LIN {X 0,Y 503.451,Z 205.902,A -85,B 0,C 180,E1 23460.888,E2 23460.888} C_VEL
LIN {X 0,Y 500.034,Z 203.731,A -85,B 0,C 180,E1 23459.638,E2 23459.638} C_VEL
LIN {X 0,Y 498.269,Z 200.894,A -85,B 0,C 180,E1 23458.928,E2 23458.928} C_VEL
LIN {X 0,Y 497.928,Z 199.39,A -85,B 0,C 180,E1 23458.464,E2 23458.464} C_VEL
LIN {X 0,Y 497.845,Z 199.153,A -85,B 0,C 180,E1 23455.087,E2 23455.087} C_VEL
LIN {X 0,Y 497.839,Z 199.158,A -85,B 0,C 180,E1 23451.564,E2 23451.564} C_VEL
LIN {X 0,Y 497.875,Z 199.15,A -85,B 0,C 180,E1 23448.167,E2 23448.167} C_VEL
LIN {X 0,Y 497.889,Z 199.152,A -85,B 0,C 180,E1 23444.66,E2 23444.66} C_VEL
LIN {X 0,Y 497.848,Z 199.155,A -85,B 0,C 180,E1 23441.206,E2 23441.206} C_VEL
LIN {X 0,Y 497.838,Z 199.151,A -85,B 0,C 180,E1 23437.7,E2 23437.7} C_VEL
LIN {X 0,Y 497.857,Z 199.101,A -85,B 0,C 180,E1 23434.219,E2 23434.219} C_VEL
LIN {X 0,Y 497.897,Z 199.14,A -85,B 0,C 180,E1 23430.751,E2 23430.751} C_VEL
LIN {X 0,Y 497.838,Z 199.082,A -85,B 0,C 180,E1 23427.383,E2 23427.383} C_VEL
LIN {X 0,Y 497.842,Z 199.154,A -85,B 0,C 180,E1 23423.936,E2 23423.936} C_VEL
LIN {X 0,Y 497.884,Z 199.137,A -85,B 0,C 180,E1 23420.576,E2 23420.576} C_VEL
LIN {X 0,Y 497.878,Z 199.13,A -85,B 0,C 180,E1 23417.05,E2 23417.05} C_VEL
LIN {X 0,Y 497.837,Z 199.149,A -85,B 0,C 180,E1 23413.71,E2 23413.71} C_VEL
LIN {X 0,Y 497.845,Z 199.151,A -85,B 0,C 180,E1 23410.18,E2 23410.18} C_VEL
LIN {X 0,Y 497.891,Z 199.129,A -85,B 0,C 180,E1 23406.805,E2 23406.805} C_VEL
LIN {X 0,Y 497.864,Z 199.14,A -85,B 0,C 180,E1 23403.339,E2 23403.339} C_VEL
LIN {X 0,Y 497.837,Z 199.152,A -85,B 0,C 180,E1 23400,E2 23400} C_VEL
LIN {X 0,Y 497.853,Z 199.133,A -85,B 0,C 180,E1 23396.546,E2 23396.546} C_VEL
LIN {X 0,Y 497.907,Z 199.128,A -85,B 0,C 180,E1 23393.079,E2 23393.079} C_VEL
LIN {X 0,Y 497.859,Z 199.15,A -85,B 0,C 180,E1 23389.586,E2 23389.586} C_VEL
LIN {X 0,Y 497.837,Z 199.145,A -85,B 0,C 180,E1 23386.172,E2 23386.172} C_VEL
LIN {X 0,Y 497.867,Z 199.132,A -85,B 0,C 180,E1 23382.829,E2 23382.829} C_VEL
LIN {X 0,Y 497.897,Z 199.142,A -85,B 0,C 180,E1 23379.301,E2 23379.301} C_VEL
LIN {X 0,Y 497.849,Z 199.152,A -85,B 0,C 180,E1 23375.939,E2 23375.939} C_VEL
LIN {X 0,Y 497.836,Z 199.091,A -85,B 0,C 180,E1 23372.487,E2 23372.487} C_VEL
LIN {X 0,Y 497.889,Z 199.132,A -85,B 0,C 180,E1 23369.196,E2 23369.196} C_VEL
LIN {X 0,Y 497.862,Z 199.118,A -85,B 0,C 180,E1 23365.782,E2 23365.782} C_VEL
LIN {X 0,Y 497.841,Z 199.156,A -85,B 0,C 180,E1 23362.369,E2 23362.369} C_VEL
LIN {X 0,Y 497.849,Z 199.132,A -85,B 0,C 180,E1 23358.856,E2 23358.856} C_VEL
LIN {X 0,Y 497.893,Z 199.121,A -85,B 0,C 180,E1 23355.465,E2 23355.465} C_VEL
LIN {X 0,Y 497.941,Z 199.447,A -85,B 0,C 180,E1 23353.525,E2 23353.525} C_VEL
LIN {X 0,Y 504.165,Z 217.265,A -85,B 0,C 180,E1 23350.484,E2 23350.484} C_VEL
LIN {X 0,Y 505.158,Z 220.046,A -85,B 0,C 180,E1 23350.091,E2 23350.091} C_VEL
LIN {X 0,Y 517.105,Z 241.444,A -85,B 0,C 180,E1 23348.608,E2 23348.608} C_VEL
LIN {X 0,Y 529.238,Z 265.386,A -85,B 0,C 180,E1 23347.173,E2 23347.173} C_VEL
LIN {X 0,Y 531.195,Z 274.082,A -85,B 0,C 180,E1 23346.87,E2 23346.87} C_VEL
LIN {X 0,Y 527.525,Z 417.717,A -85,B 0,C 180,E1 23344.805,E2 23344.805} C_VEL
LIN {X 0,Y 524.676,Z 523.398,A -85,B 0,C 180,E1 23343.275,E2 23343.275} C_VEL
LIN {X 0,Y 523.631,Z 541.9,A -85,B 0,C 180,E1 23342.893,E2 23342.893} C_VEL
LIN {X 0,Y 521.95,Z 563.753,A -85,B 0,C 180,E1 23342.271,E2 23342.271} C_VEL
LIN {X 0,Y 519.848,Z 584.783,A -85,B 0,C 180,E1 23341.453,E2 23341.453} C_VEL
LIN {X 0,Y 517.885,Z 601.843,A -85,B 0,C 180,E1 23340.64,E2 23340.64} C_VEL
LIN {X 0,Y 515.872,Z 617.714,A -85,B 0,C 180,E1 23339.744,E2 23339.744} C_VEL
LIN {X 0,Y 513.731,Z 633.164,A -85,B 0,C 180,E1 23338.73,E2 23338.73} C_VEL
LIN {X 0,Y 511.543,Z 648.153,A -85,B 0,C 180,E1 23337.593,E2 23337.593} C_VEL
LIN {X 0,Y 509.129,Z 663.894,A -85,B 0,C 180,E1 23336.22,E2 23336.22} C_VEL
LIN {X 0,Y 506.185,Z 682.494,A -85,B 0,C 180,E1 23334.302,E2 23334.302} C_VEL
LIN {X 0,Y 504.116,Z 695.494,A -85,B 0,C 180,E1 23332.734,E2 23332.734} C_VEL
LIN {X 0,Y 502.283,Z 707.263,A -85,B 0,C 180,E1 23331.116,E2 23331.116} C_VEL
LIN {X 0,Y 500.73,Z 717.761,A -85,B 0,C 180,E1 23329.477,E2 23329.477} C_VEL
LIN {X 0,Y 499.357,Z 727.653,A -85,B 0,C 180,E1 23327.717,E2 23327.717} C_VEL
LIN {X 0,Y 498.274,Z 736.294,A -85,B 0,C 180,E1 23325.955,E2 23325.955} C_VEL
LIN {X 0,Y 497.385,Z 744.272,A -85,B 0,C 180,E1 23324.076,E2 23324.076} C_VEL
LIN {X 0,Y 496.688,Z 751.974,A -85,B 0,C 180,E1 23321.936,E2 23321.936} C_VEL
LIN {X 0,Y 496.191,Z 759.575,A -85,B 0,C 180,E1 23319.276,E2 23319.276} C_VEL
LIN {X 0,Y 495.993,Z 764.333,A -85,B 0,C 180,E1 23317.063,E2 23317.063} C_VEL
LIN {X 0,Y 495.929,Z 767.482,A -85,B 0,C 180,E1 23315.089,E2 23315.089} C_VEL
LIN {X 0,Y 495.921,Z 769.593,A -85,B 0,C 180,E1 23313.12,E2 23313.12} C_VEL
LIN {X 0,Y 495.93,Z 770.688,A -85,B 0,C 180,E1 23311.155,E2 23311.155} C_VEL
LIN {X 0,Y 495.934,Z 770.776,A -85,B 0,C 180,E1 23309.191,E2 23309.191} C_VEL
LIN {X 0,Y 495.925,Z 769.858,A -85,B 0,C 180,E1 23307.227,E2 23307.227} C_VEL
LIN {X 0,Y 495.926,Z 767.925,A -85,B 0,C 180,E1 23305.259,E2 23305.259} C_VEL
LIN {X 0,Y 495.976,Z 764.957,A -85,B 0,C 180,E1 23303.286,E2 23303.286} C_VEL
LIN {X 0,Y 496.12,Z 760.924,A -85,B 0,C 180,E1 23301.307,E2 23301.307} C_VEL
LIN {X 0,Y 496.417,Z 755.784,A -85,B 0,C 180,E1 23299.322,E2 23299.322} C_VEL
LIN {X 0,Y 496.898,Z 749.477,A -85,B 0,C 180,E1 23297.332,E2 23297.332} C_VEL
LIN {X 0,Y 497.688,Z 741.461,A -85,B 0,C 180,E1 23295.219,E2 23295.219} C_VEL
LIN {X 0,Y 499.12,Z 729.508,A -85,B 0,C 180,E1 23292.635,E2 23292.635} C_VEL
LIN {X 0,Y 500.531,Z 719.165,A -85,B 0,C 180,E1 23290.757,E2 23290.757} C_VEL
LIN {X 0,Y 502.164,Z 708.055,A -85,B 0,C 180,E1 23289,E2 23289} C_VEL
LIN {X 0,Y 503.847,Z 697.151,A -85,B 0,C 180,E1 23287.483,E2 23287.483} C_VEL
LIN {X 0,Y 505.805,Z 684.805,A -85,B 0,C 180,E1 23285.966,E2 23285.966} C_VEL
LIN {X 0,Y 507.923,Z 671.506,A -85,B 0,C 180,E1 23284.528,E2 23284.528} C_VEL
LIN {X 0,Y 510.51,Z 655.066,A -85,B 0,C 180,E1 23282.978,E2 23282.978} C_VEL
LIN {X 0,Y 513.382,Z 635.707,A -85,B 0,C 180,E1 23281.45,E2 23281.45} C_VEL
LIN {X 0,Y 515.631,Z 619.555,A -85,B 0,C 180,E1 23280.369,E2 23280.369} C_VEL
LIN {X 0,Y 517.632,Z 603.968,A -85,B 0,C 180,E1 23279.472,E2 23279.472} C_VEL
LIN {X 0,Y 519.49,Z 588.073,A -85,B 0,C 180,E1 23278.694,E2 23278.694} C_VEL
LIN {X 0,Y 521.153,Z 571.933,A -85,B 0,C 180,E1 23278.031,E2 23278.031} C_VEL
LIN {X 0,Y 522.647,Z 554.985,A -85,B 0,C 180,E1 23277.463,E2 23277.463} C_VEL
LIN {X 0,Y 523.887,Z 537.918,A -85,B 0,C 180,E1 23277.015,E2 23277.015} C_VEL
LIN {X 0,Y 524.82,Z 519.908,A -85,B 0,C 180,E1 23276.666,E2 23276.666} C_VEL
LIN {X 0,Y 531.341,Z 274.821,A -85,B 0,C 180,E1 23273.154,E2 23273.154} C_VEL
LIN {X 0,Y 529.324,Z 265.566,A -85,B 0,C 180,E1 23272.837,E2 23272.837} C_VEL
LIN {X 0,Y 517.446,Z 242.108,A -85,B 0,C 180,E1 23271.433,E2 23271.433} C_VEL
LIN {X 0,Y 507.217,Z 223.795,A -85,B 0,C 180,E1 23270.182,E2 23270.182} C_VEL
LIN {X 0,Y 504.803,Z 219.133,A -85,B 0,C 180,E1 23269.817,E2 23269.817} C_VEL
LIN {X 0,Y 499.451,Z 204.085,A -85,B 0,C 180,E1 23267.284,E2 23267.284} C_VEL
LIN {X 0,Y 497.906,Z 199.22,A -85,B 0,C 180,E1 23266.403,E2 23266.403} C_VEL
LIN {X 0,Y 497.87,Z 199.143,A -85,B 0,C 180,E1 23262.866,E2 23262.866} C_VEL
LIN {X 0,Y 497.835,Z 199.125,A -85,B 0,C 180,E1 23259.543,E2 23259.543} C_VEL
LIN {X 0,Y 497.862,Z 199.128,A -85,B 0,C 180,E1 23256.172,E2 23256.172} C_VEL
LIN {X 0,Y 497.893,Z 199.143,A -85,B 0,C 180,E1 23252.699,E2 23252.699} C_VEL
LIN {X 0,Y 497.841,Z 199.096,A -85,B 0,C 180,E1 23249.345,E2 23249.345} C_VEL
LIN {X 0,Y 497.839,Z 199.133,A -85,B 0,C 180,E1 23245.839,E2 23245.839} C_VEL
LIN {X 0,Y 497.872,Z 199.132,A -85,B 0,C 180,E1 23242.432,E2 23242.432} C_VEL
LIN {X 0,Y 497.886,Z 199.14,A -85,B 0,C 180,E1 23238.956,E2 23238.956} C_VEL
LIN {X 0,Y 497.842,Z 199.149,A -85,B 0,C 180,E1 23235.613,E2 23235.613} C_VEL
LIN {X 0,Y 497.839,Z 199.14,A -85,B 0,C 180,E1 23232.045,E2 23232.045} C_VEL
LIN {X 0,Y 497.877,Z 199.128,A -85,B 0,C 180,E1 23228.663,E2 23228.663} C_VEL
LIN {X 0,Y 497.868,Z 199.152,A -85,B 0,C 180,E1 23225.301,E2 23225.301} C_VEL
LIN {X 0,Y 497.839,Z 199.144,A -85,B 0,C 180,E1 23221.842,E2 23221.842} C_VEL
LIN {X 0,Y 497.839,Z 199.133,A -85,B 0,C 180,E1 23218.274,E2 23218.274} C_VEL
LIN {X 0,Y 497.878,Z 199.148,A -85,B 0,C 180,E1 23214.815,E2 23214.815} C_VEL
LIN {X 0,Y 497.865,Z 199.141,A -85,B 0,C 180,E1 23211.453,E2 23211.453} C_VEL
LIN {X 0,Y 497.836,Z 199.134,A -85,B 0,C 180,E1 23208.061,E2 23208.061} C_VEL
LIN {X 0,Y 497.848,Z 199.148,A -85,B 0,C 180,E1 23204.56,E2 23204.56} C_VEL
LIN {X 0,Y 497.895,Z 199.148,A -85,B 0,C 180,E1 23201.136,E2 23201.136} C_VEL
LIN {X 0,Y 497.858,Z 199.138,A -85,B 0,C 180,E1 23197.692,E2 23197.692} C_VEL
LIN {X 0,Y 497.836,Z 199.121,A -85,B 0,C 180,E1 23194.289,E2 23194.289} C_VEL
LIN {X 0,Y 497.847,Z 199.1,A -85,B 0,C 180,E1 23190.788,E2 23190.788} C_VEL
LIN {X 0,Y 497.895,Z 199.139,A -85,B 0,C 180,E1 23187.438,E2 23187.438} C_VEL
LIN {X 0,Y 497.845,Z 199.102,A -85,B 0,C 180,E1 23183.951,E2 23183.951} C_VEL
LIN {X 0,Y 497.841,Z 199.155,A -85,B 0,C 180,E1 23180.604,E2 23180.604} C_VEL
LIN {X 0,Y 497.882,Z 199.153,A -85,B 0,C 180,E1 23177.25,E2 23177.25} C_VEL
LIN {X 0,Y 497.869,Z 199.151,A -85,B 0,C 180,E1 23173.851,E2 23173.851} C_VEL
LIN {X 0,Y 497.842,Z 199.154,A -85,B 0,C 180,E1 23170.429,E2 23170.429} C_VEL
LIN {X 0,Y 497.846,Z 199.155,A -85,B 0,C 180,E1 23166.901,E2 23166.901} C_VEL
LIN {X 0,Y 497.892,Z 199.148,A -85,B 0,C 180,E1 23163.518,E2 23163.518} C_VEL
LIN {X 0,Y 497.927,Z 199.388,A -85,B 0,C 180,E1 23161.536,E2 23161.536} C_VEL
LIN {X 0,Y 498.266,Z 200.884,A -85,B 0,C 180,E1 23161.072,E2 23161.072} C_VEL
LIN {X 0,Y 500.031,Z 203.728,A -85,B 0,C 180,E1 23160.361,E2 23160.361} C_VEL
LIN {X 0,Y 503.944,Z 206.453,A -85,B 0,C 180,E1 23158.922,E2 23158.922} C_VEL
LIN {X 0,Y 505.99,Z 209.837,A -85,B 0,C 180,E1 23158.05,E2 23158.05} C_VEL
LIN {X 0,Y 508.653,Z 212.064,A -85,B 0,C 180,E1 23157.002,E2 23157.002} C_VEL
LIN {X 0,Y 510.463,Z 213.14,A -85,B 0,C 180,E1 23156.272,E2 23156.272} C_VEL
LIN {X 0,Y 512.499,Z 216.574,A -85,B 0,C 180,E1 23155.332,E2 23155.332} C_VEL
LIN {X 0,Y 515.184,Z 218.79,A -85,B 0,C 180,E1 23154.171,E2 23154.171} C_VEL
LIN {X 0,Y 517.234,Z 220.098,A -85,B 0,C 180,E1 23153.262,E2 23153.262} C_VEL
LIN {X 0,Y 519.49,Z 223.636,A -85,B 0,C 180,E1 23152.101,E2 23152.101} C_VEL
LIN {X 0,Y 522.505,Z 225.999,A -85,B 0,C 180,E1 23150.614,E2 23150.614} C_VEL
LIN {X 0,Y 524.11,Z 226.919,A -85,B 0,C 180,E1 23149.797,E2 23149.797} C_VEL
LIN {X 0,Y 526.402,Z 230.454,A -85,B 0,C 180,E1 23148.434,E2 23148.434} C_VEL
LIN {X 0,Y 529.142,Z 232.753,A -85,B 0,C 180,E1 23146.803,E2 23146.803} C_VEL
LIN {X 0,Y 531.496,Z 234.088,A -85,B 0,C 180,E1 23145.324,E2 23145.324} C_VEL
LIN {X 0,Y 533.417,Z 237.302,A -85,B 0,C 180,E1 23143.834,E2 23143.834} C_VEL
LIN {X 0,Y 535.894,Z 239.476,A -85,B 0,C 180,E1 23141.842,E2 23141.842} C_VEL
LIN {X 0,Y 538.639,Z 240.894,A -85,B 0,C 180,E1 23139.293,E2 23139.293} C_VEL
LIN {X 0,Y 539.733,Z 242.544,A -85,B 0,C 180,E1 23137.878,E2 23137.878} C_VEL
LIN {X 0,Y 541.029,Z 244.652,A -85,B 0,C 180,E1 23135.727,E2 23135.727} C_VEL
LIN {X 0,Y 542.124,Z 245.772,A -85,B 0,C 180,E1 23133.171,E2 23133.171} C_VEL
LIN {X 0,Y 542.593,Z 246.138,A -85,B 0,C 180,E1 23130.633,E2 23130.633} C_VEL
LIN {X 0,Y 542.445,Z 245.986,A -85,B 0,C 180,E1 23128.099,E2 23128.099} C_VEL
LIN {X 0,Y 541.709,Z 245.347,A -85,B 0,C 180,E1 23125.66,E2 23125.66} C_VEL
LIN {X 0,Y 540.629,Z 243.992,A -85,B 0,C 180,E1 23123.523,E2 23123.523} C_VEL
LIN {X 0,Y 539.601,Z 242.211,A -85,B 0,C 180,E1 23121.905,E2 23121.905} C_VEL
LIN {X 0,Y 538.194,Z 240.612,A -85,B 0,C 180,E1 23120.268,E2 23120.268} C_VEL
LIN {X 0,Y 535.66,Z 239.296,A -85,B 0,C 180,E1 23117.934,E2 23117.934} C_VEL
LIN {X 0,Y 533.198,Z 237.042,A -85,B 0,C 180,E1 23116.003,E2 23116.003} C_VEL
LIN {X 0,Y 532.754,Z 236.42,A -85,B 0,C 180,E1 23115.654,E2 23115.654} C_VEL
LIN {X 0,Y 531.754,Z 235.905,A -85,B 0,C 180,E1 23114.949,E2 23114.949} C_VEL
LIN {X 0,Y 529.6,Z 237.547,A -85,B 0,C 180,E1 23113.775,E2 23113.775} C_VEL
LIN {X 0,Y 527.161,Z 239.389,A -85,B 0,C 180,E1 23112.536,E2 23112.536} C_VEL
LIN {X 0,Y 525.922,Z 239.086,A -85,B 0,C 180,E1 23111.882,E2 23111.882} C_VEL
LIN {X 0,Y 523.308,Z 235.692,A -85,B 0,C 180,E1 23110.352,E2 23110.352} C_VEL
LIN {X 0,Y 522.483,Z 234.359,A -85,B 0,C 180,E1 23109.853,E2 23109.853} C_VEL
LIN {X 0,Y 519.054,Z 232.276,A -85,B 0,C 180,E1 23108.177,E2 23108.177} C_VEL
LIN {X 0,Y 516.336,Z 228.871,A -85,B 0,C 180,E1 23106.825,E2 23106.825} C_VEL
LIN {X 0,Y 515.278,Z 227.326,A -85,B 0,C 180,E1 23106.32,E2 23106.32} C_VEL
LIN {X 0,Y 511.735,Z 225.034,A -85,B 0,C 180,E1 23104.793,E2 23104.793} C_VEL
LIN {X 0,Y 509.276,Z 221.656,A -85,B 0,C 180,E1 23103.694,E2 23103.694} C_VEL
LIN {X 0,Y 508.559,Z 220.481,A -85,B 0,C 180,E1 23103.371,E2 23103.371} C_VEL
LIN {X 0,Y 505.312,Z 218.416,A -85,B 0,C 180,E1 23102.101,E2 23102.101} C_VEL
LIN {X 0,Y 502.758,Z 215.081,A -85,B 0,C 180,E1 23101.054,E2 23101.054} C_VEL
LIN {X 0,Y 501.761,Z 213.558,A -85,B 0,C 180,E1 23100.649,E2 23100.649} C_VEL
LIN {X 0,Y 498.421,Z 211.369,A -85,B 0,C 180,E1 23099.438,E2 23099.438} C_VEL
LIN {X 0,Y 496.347,Z 208.221,A -85,B 0,C 180,E1 23098.611,E2 23098.611} C_VEL
LIN {X 0,Y 495.458,Z 206.833,A -85,B 0,C 180,E1 23098.281,E2 23098.281} C_VEL
LIN {X 0,Y 492.073,Z 204.698,A -85,B 0,C 180,E1 23097.118,E2 23097.118} C_VEL
LIN {X 0,Y 490.363,Z 201.853,A -85,B 0,C 180,E1 23096.483,E2 23096.483} C_VEL
LIN {X 0,Y 490.01,Z 200.59,A -85,B 0,C 180,E1 23096.151,E2 23096.151} C_VEL
LIN {X 0,Y 489.901,Z 200.144,A -85,B 0,C 180,E1 23095.294,E2 23095.294} C_VEL
LIN {X 0,Y 489.908,Z 200.143,A -85,B 0,C 180,E1 23091.793,E2 23091.793} C_VEL
LIN {X 0,Y 489.962,Z 200.139,A -85,B 0,C 180,E1 23088.459,E2 23088.459} C_VEL
LIN {X 0,Y 489.925,Z 200.143,A -85,B 0,C 180,E1 23084.92,E2 23084.92} C_VEL
LIN {X 0,Y 489.901,Z 200.144,A -85,B 0,C 180,E1 23081.501,E2 23081.501} C_VEL
LIN {X 0,Y 489.913,Z 200.141,A -85,B 0,C 180,E1 23078.029,E2 23078.029} C_VEL
LIN {X 0,Y 489.945,Z 200.08,A -85,B 0,C 180,E1 23074.566,E2 23074.566} C_VEL
LIN {X 0,Y 489.924,Z 200.14,A -85,B 0,C 180,E1 23071.088,E2 23071.088} C_VEL
LIN {X 0,Y 489.892,Z 200.068,A -85,B 0,C 180,E1 23067.663,E2 23067.663} C_VEL
LIN {X 0,Y 489.909,Z 200.143,A -85,B 0,C 180,E1 23064.092,E2 23064.092} C_VEL
LIN {X 0,Y 489.954,Z 200.123,A -85,B 0,C 180,E1 23060.674,E2 23060.674} C_VEL
LIN {X 0,Y 489.924,Z 200.121,A -85,B 0,C 180,E1 23057.213,E2 23057.213} C_VEL
LIN {X 0,Y 489.898,Z 200.138,A -85,B 0,C 180,E1 23053.816,E2 23053.816} C_VEL
LIN {X 0,Y 489.915,Z 200.14,A -85,B 0,C 180,E1 23050.347,E2 23050.347} C_VEL
LIN {X 0,Y 489.964,Z 200.115,A -85,B 0,C 180,E1 23046.915,E2 23046.915} C_VEL
LIN {X 0,Y 489.92,Z 200.13,A -85,B 0,C 180,E1 23043.393,E2 23043.393} C_VEL
LIN {X 0,Y 489.899,Z 200.141,A -85,B 0,C 180,E1 23040,E2 23040} C_VEL
LIN {X 0,Y 489.91,Z 200.122,A -85,B 0,C 180,E1 23036.49,E2 23036.49} C_VEL
LIN {X 0,Y 489.967,Z 200.117,A -85,B 0,C 180,E1 23033.085,E2 23033.085} C_VEL
LIN {X 0,Y 489.924,Z 200.139,A -85,B 0,C 180,E1 23029.535,E2 23029.535} C_VEL
LIN {X 0,Y 489.9,Z 200.134,A -85,B 0,C 180,E1 23026.064,E2 23026.064} C_VEL
LIN {X 0,Y 489.908,Z 200.121,A -85,B 0,C 180,E1 23022.541,E2 23022.541} C_VEL
LIN {X 0,Y 489.95,Z 200.128,A -85,B 0,C 180,E1 23019.075,E2 23019.075} C_VEL
LIN {X 0,Y 489.93,Z 200.142,A -85,B 0,C 180,E1 23015.653,E2 23015.653} C_VEL
LIN {X 0,Y 489.894,Z 200.076,A -85,B 0,C 180,E1 23012.267,E2 23012.267} C_VEL
LIN {X 0,Y 489.912,Z 200.135,A -85,B 0,C 180,E1 23008.765,E2 23008.765} C_VEL
LIN {X 0,Y 489.945,Z 200.098,A -85,B 0,C 180,E1 23005.292,E2 23005.292} C_VEL
LIN {X 0,Y 489.931,Z 200.133,A -85,B 0,C 180,E1 23001.779,E2 23001.779} C_VEL
LIN {X 0,Y 489.904,Z 200.135,A -85,B 0,C 180,E1 22998.323,E2 22998.323} C_VEL
LIN {X 0,Y 489.903,Z 200.123,A -85,B 0,C 180,E1 22994.743,E2 22994.743} C_VEL
LIN {X 0,Y 489.958,Z 200.471,A -85,B 0,C 180,E1 22994.228,E2 22994.228} C_VEL
LIN {X 0,Y 495.655,Z 216.642,A -85,B 0,C 180,E1 22991.371,E2 22991.371} C_VEL
LIN {X 0,Y 496.799,Z 219.731,A -85,B 0,C 180,E1 22990.908,E2 22990.908} C_VEL
LIN {X 0,Y 509.038,Z 241.244,A -85,B 0,C 180,E1 22989.336,E2 22989.336} C_VEL
LIN {X 0,Y 521.009,Z 264.31,A -85,B 0,C 180,E1 22987.877,E2 22987.877} C_VEL
LIN {X 0,Y 523.811,Z 270.751,A -85,B 0,C 180,E1 22987.531,E2 22987.531} C_VEL
LIN {X 0,Y 524.883,Z 277.55,A -85,B 0,C 180,E1 22987.327,E2 22987.327} C_VEL
LIN {X 0,Y 518.017,Z 522.61,A -85,B 0,C 180,E1 22983.772,E2 22983.772} C_VEL
LIN {X 0,Y 516.991,Z 540.545,A -85,B 0,C 180,E1 22983.403,E2 22983.403} C_VEL
LIN {X 0,Y 515.489,Z 559.735,A -85,B 0,C 180,E1 22982.868,E2 22982.868} C_VEL
LIN {X 0,Y 513.182,Z 582.921,A -85,B 0,C 180,E1 22981.998,E2 22981.998} C_VEL
LIN {X 0,Y 511.083,Z 600.604,A -85,B 0,C 180,E1 22981.158,E2 22981.158} C_VEL
LIN {X 0,Y 508.983,Z 616.616,A -85,B 0,C 180,E1 22980.253,E2 22980.253} C_VEL
LIN {X 0,Y 506.745,Z 632.18,A -85,B 0,C 180,E1 22979.228,E2 22979.228} C_VEL
LIN {X 0,Y 504.56,Z 646.608,A -85,B 0,C 180,E1 22978.132,E2 22978.132} C_VEL
LIN {X 0,Y 502.293,Z 660.825,A -85,B 0,C 180,E1 22976.898,E2 22976.898} C_VEL
LIN {X 0,Y 500.016,Z 674.694,A -85,B 0,C 180,E1 22975.523,E2 22975.523} C_VEL
LIN {X 0,Y 497.381,Z 690.681,A -85,B 0,C 180,E1 22973.704,E2 22973.704} C_VEL
LIN {X 0,Y 494.882,Z 705.762,A -85,B 0,C 180,E1 22971.656,E2 22971.656} C_VEL
LIN {X 0,Y 493.131,Z 716.881,A -85,B 0,C 180,E1 22969.913,E2 22969.913} C_VEL
LIN {X 0,Y 491.664,Z 726.855,A -85,B 0,C 180,E1 22968.126,E2 22968.126} C_VEL
LIN {X 0,Y 490.496,Z 735.574,A -85,B 0,C 180,E1 22966.336,E2 22966.336} C_VEL
LIN {X 0,Y 489.54,Z 743.626,A -85,B 0,C 180,E1 22964.427,E2 22964.427} C_VEL
LIN {X 0,Y 488.858,Z 750.498,A -85,B 0,C 180,E1 22962.52,E2 22962.52} C_VEL
LIN {X 0,Y 488.383,Z 756.607,A -85,B 0,C 180,E1 22960.497,E2 22960.497} C_VEL
LIN {X 0,Y 488.07,Z 762.367,A -85,B 0,C 180,E1 22958.125,E2 22958.125} C_VEL
LIN {X 0,Y 487.939,Z 767.011,A -85,B 0,C 180,E1 22955.408,E2 22955.408} C_VEL
LIN {X 0,Y 487.923,Z 769.33,A -85,B 0,C 180,E1 22953.289,E2 22953.289} C_VEL
LIN {X 0,Y 487.929,Z 770.484,A -85,B 0,C 180,E1 22951.291,E2 22951.291} C_VEL
LIN {X 0,Y 487.935,Z 770.631,A -85,B 0,C 180,E1 22949.296,E2 22949.296} C_VEL
LIN {X 0,Y 487.927,Z 769.771,A -85,B 0,C 180,E1 22947.299,E2 22947.299} C_VEL
LIN {X 0,Y 487.927,Z 767.897,A -85,B 0,C 180,E1 22945.299,E2 22945.299} C_VEL
LIN {X 0,Y 487.976,Z 764.989,A -85,B 0,C 180,E1 22943.294,E2 22943.294} C_VEL
LIN {X 0,Y 488.122,Z 761.018,A -85,B 0,C 180,E1 22941.282,E2 22941.282} C_VEL
LIN {X 0,Y 488.429,Z 755.94,A -85,B 0,C 180,E1 22939.265,E2 22939.265} C_VEL
LIN {X 0,Y 488.912,Z 749.894,A -85,B 0,C 180,E1 22937.3,E2 22937.3} C_VEL
LIN {X 0,Y 489.645,Z 742.689,A -85,B 0,C 180,E1 22935.334,E2 22935.334} C_VEL
LIN {X 0,Y 490.733,Z 733.77,A -85,B 0,C 180,E1 22933.266,E2 22933.266} C_VEL
LIN {X 0,Y 492.514,Z 721.091,A -85,B 0,C 180,E1 22930.801,E2 22930.801} C_VEL
LIN {X 0,Y 494.38,Z 708.868,A -85,B 0,C 180,E1 22928.81,E2 22928.81} C_VEL
LIN {X 0,Y 496.16,Z 697.863,A -85,B 0,C 180,E1 22927.24,E2 22927.24} C_VEL
LIN {X 0,Y 498.256,Z 685.24,A -85,B 0,C 180,E1 22925.655,E2 22925.655} C_VEL
LIN {X 0,Y 500.384,Z 672.45,A -85,B 0,C 180,E1 22924.243,E2 22924.243} C_VEL
LIN {X 0,Y 502.709,Z 658.244,A -85,B 0,C 180,E1 22922.865,E2 22922.865} C_VEL
LIN {X 0,Y 505.48,Z 640.863,A -85,B 0,C 180,E1 22921.404,E2 22921.404} C_VEL
LIN {X 0,Y 508.36,Z 621.219,A -85,B 0,C 180,E1 22920.032,E2 22920.032} C_VEL
LIN {X 0,Y 510.547,Z 604.927,A -85,B 0,C 180,E1 22919.072,E2 22919.072} C_VEL
LIN {X 0,Y 512.538,Z 588.6,A -85,B 0,C 180,E1 22918.257,E2 22918.257} C_VEL
LIN {X 0,Y 514.34,Z 571.757,A -85,B 0,C 180,E1 22917.556,E2 22917.556} C_VEL
LIN {X 0,Y 515.899,Z 554.695,A -85,B 0,C 180,E1 22916.979,E2 22916.979} C_VEL
LIN {X 0,Y 517.185,Z 537.595,A -85,B 0,C 180,E1 22916.528,E2 22916.528} C_VEL
LIN {X 0,Y 518.157,Z 519.322,A -85,B 0,C 180,E1 22916.172,E2 22916.172} C_VEL
LIN {X 0,Y 524.879,Z 276.252,A -85,B 0,C 180,E1 22912.651,E2 22912.651} C_VEL
LIN {X 0,Y 523.288,Z 269.108,A -85,B 0,C 180,E1 22912.398,E2 22912.398} C_VEL
LIN {X 0,Y 511.077,Z 244.975,A -85,B 0,C 180,E1 22910.916,E2 22910.916} C_VEL
LIN {X 0,Y 499.266,Z 223.903,A -85,B 0,C 180,E1 22909.423,E2 22909.423} C_VEL
LIN {X 0,Y 496.42,Z 218.848,A -85,B 0,C 180,E1 22908.998,E2 22908.998} C_VEL
LIN {X 0,Y 491.01,Z 203.253,A -85,B 0,C 180,E1 22906.296,E2 22906.296} C_VEL
LIN {X 0,Y 489.91,Z 200.189,A -85,B 0,C 180,E1 22905.666,E2 22905.666} C_VEL
LIN {X 0,Y 489.936,Z 200.142,A -85,B 0,C 180,E1 22902.206,E2 22902.206} C_VEL
LIN {X 0,Y 489.96,Z 200.12,A -85,B 0,C 180,E1 22898.644,E2 22898.644} C_VEL
LIN {X 0,Y 489.912,Z 200.102,A -85,B 0,C 180,E1 22895.138,E2 22895.138} C_VEL
LIN {X 0,Y 489.903,Z 200.142,A -85,B 0,C 180,E1 22891.637,E2 22891.637} C_VEL
LIN {X 0,Y 489.908,Z 200.071,A -85,B 0,C 180,E1 22888.13,E2 22888.13} C_VEL
LIN {X 0,Y 489.957,Z 200.134,A -85,B 0,C 180,E1 22884.731,E2 22884.731} C_VEL
LIN {X 0,Y 489.913,Z 200.126,A -85,B 0,C 180,E1 22881.303,E2 22881.303} C_VEL
LIN {X 0,Y 489.9,Z 200.12,A -85,B 0,C 180,E1 22877.828,E2 22877.828} C_VEL
LIN {X 0,Y 489.914,Z 200.131,A -85,B 0,C 180,E1 22874.298,E2 22874.298} C_VEL
LIN {X 0,Y 489.952,Z 200.135,A -85,B 0,C 180,E1 22870.822,E2 22870.822} C_VEL
LIN {X 0,Y 489.917,Z 200.119,A -85,B 0,C 180,E1 22867.361,E2 22867.361} C_VEL
LIN {X 0,Y 489.898,Z 200.133,A -85,B 0,C 180,E1 22863.979,E2 22863.979} C_VEL
LIN {X 0,Y 489.915,Z 200.142,A -85,B 0,C 180,E1 22860.468,E2 22860.468} C_VEL
LIN {X 0,Y 489.949,Z 200.119,A -85,B 0,C 180,E1 22857.015,E2 22857.015} C_VEL
LIN {X 0,Y 489.915,Z 200.126,A -85,B 0,C 180,E1 22853.555,E2 22853.555} C_VEL
LIN {X 0,Y 489.9,Z 200.142,A -85,B 0,C 180,E1 22850.128,E2 22850.128} C_VEL
LIN {X 0,Y 489.918,Z 200.131,A -85,B 0,C 180,E1 22846.666,E2 22846.666} C_VEL
LIN {X 0,Y 489.951,Z 200.119,A -85,B 0,C 180,E1 22843.277,E2 22843.277} C_VEL
LIN {X 0,Y 489.912,Z 200.139,A -85,B 0,C 180,E1 22839.823,E2 22839.823} C_VEL
LIN {X 0,Y 489.901,Z 200.143,A -85,B 0,C 180,E1 22836.292,E2 22836.292} C_VEL
LIN {X 0,Y 489.91,Z 200.07,A -85,B 0,C 180,E1 22832.795,E2 22832.795} C_VEL
LIN {X 0,Y 489.966,Z 200.126,A -85,B 0,C 180,E1 22829.324,E2 22829.324} C_VEL
LIN {X 0,Y 489.913,Z 200.09,A -85,B 0,C 180,E1 22825.857,E2 22825.857} C_VEL
LIN {X 0,Y 489.899,Z 200.136,A -85,B 0,C 180,E1 22822.354,E2 22822.354} C_VEL
LIN {X 0,Y 489.913,Z 200.143,A -85,B 0,C 180,E1 22818.852,E2 22818.852} C_VEL
LIN {X 0,Y 489.952,Z 200.14,A -85,B 0,C 180,E1 22815.409,E2 22815.409} C_VEL
LIN {X 0,Y 489.933,Z 200.139,A -85,B 0,C 180,E1 22811.848,E2 22811.848} C_VEL
LIN {X 0,Y 489.9,Z 200.146,A -85,B 0,C 180,E1 22808.493,E2 22808.493} C_VEL
LIN {X 0,Y 489.91,Z 200.142,A -85,B 0,C 180,E1 22804.99,E2 22804.99} C_VEL
LIN {X 0,Y 489.956,Z 200.342,A -85,B 0,C 180,E1 22803.993,E2 22803.993} C_VEL
LIN {X 0,Y 490.307,Z 201.683,A -85,B 0,C 180,E1 22803.544,E2 22803.544} C_VEL
LIN {X 0,Y 491.956,Z 204.572,A -85,B 0,C 180,E1 22802.921,E2 22802.921} C_VEL
LIN {X 0,Y 494.818,Z 206.556,A -85,B 0,C 180,E1 22801.929,E2 22801.929} C_VEL
LIN {X 0,Y 496.06,Z 207.611,A -85,B 0,C 180,E1 22801.501,E2 22801.501} C_VEL
LIN {X 0,Y 498.022,Z 210.937,A -85,B 0,C 180,E1 22800.71,E2 22800.71} C_VEL
LIN {X 0,Y 500.893,Z 213.125,A -85,B 0,C 180,E1 22799.669,E2 22799.669} C_VEL
LIN {X 0,Y 502.22,Z 214.04,A -85,B 0,C 180,E1 22799.171,E2 22799.171} C_VEL
LIN {X 0,Y 504.483,Z 217.524,A -85,B 0,C 180,E1 22798.238,E2 22798.238} C_VEL
LIN {X 0,Y 507.499,Z 219.972,A -85,B 0,C 180,E1 22797.058,E2 22797.058} C_VEL
LIN {X 0,Y 508.891,Z 220.896,A -85,B 0,C 180,E1 22796.485,E2 22796.485} C_VEL
LIN {X 0,Y 511.269,Z 224.529,A -85,B 0,C 180,E1 22795.418,E2 22795.418} C_VEL
LIN {X 0,Y 514.35,Z 226.861,A -85,B 0,C 180,E1 22794.091,E2 22794.091} C_VEL
LIN {X 0,Y 515.772,Z 227.876,A -85,B 0,C 180,E1 22793.451,E2 22793.451} C_VEL
LIN {X 0,Y 518.223,Z 231.482,A -85,B 0,C 180,E1 22792.217,E2 22792.217} C_VEL
LIN {X 0,Y 521.433,Z 233.928,A -85,B 0,C 180,E1 22790.645,E2 22790.645} C_VEL
LIN {X 0,Y 522.805,Z 234.733,A -85,B 0,C 180,E1 22789.959,E2 22789.959} C_VEL
LIN {X 0,Y 525.228,Z 238.335,A -85,B 0,C 180,E1 22788.535,E2 22788.535} C_VEL
LIN {X 0,Y 528.09,Z 240.683,A -85,B 0,C 180,E1 22786.837,E2 22786.837} C_VEL
LIN {X 0,Y 530.357,Z 242.035,A -85,B 0,C 180,E1 22785.414,E2 22785.414} C_VEL
LIN {X 0,Y 532.316,Z 245.205,A -85,B 0,C 180,E1 22783.91,E2 22783.91} C_VEL
LIN {X 0,Y 534.886,Z 247.416,A -85,B 0,C 180,E1 22781.865,E2 22781.865} C_VEL
LIN {X 0,Y 537.641,Z 248.837,A -85,B 0,C 180,E1 22779.31,E2 22779.31} C_VEL
LIN {X 0,Y 538.796,Z 250.707,A -85,B 0,C 180,E1 22777.785,E2 22777.785} C_VEL
LIN {X 0,Y 540.296,Z 252.83,A -85,B 0,C 180,E1 22775.349,E2 22775.349} C_VEL
LIN {X 0,Y 541.303,Z 253.841,A -85,B 0,C 180,E1 22772.752,E2 22772.752} C_VEL
LIN {X 0,Y 541.665,Z 254.083,A -85,B 0,C 180,E1 22770.212,E2 22770.212} C_VEL
LIN {X 0,Y 541.41,Z 253.872,A -85,B 0,C 180,E1 22767.778,E2 22767.778} C_VEL
LIN {X 0,Y 540.525,Z 253.101,A -85,B 0,C 180,E1 22765.226,E2 22765.226} C_VEL
LIN {X 0,Y 539.177,Z 251.413,A -85,B 0,C 180,E1 22762.816,E2 22762.816} C_VEL
LIN {X 0,Y 537.731,Z 248.914,A -85,B 0,C 180,E1 22760.799,E2 22760.799} C_VEL
LIN {X 0,Y 535.004,Z 247.503,A -85,B 0,C 180,E1 22758.247,E2 22758.247} C_VEL
LIN {X 0,Y 532.408,Z 245.306,A -85,B 0,C 180,E1 22756.157,E2 22756.157} C_VEL
LIN {X 0,Y 530.515,Z 242.327,A -85,B 0,C 180,E1 22754.703,E2 22754.703} C_VEL
LIN {X 0,Y 529.319,Z 241.229,A -85,B 0,C 180,E1 22753.88,E2 22753.88} C_VEL
LIN {X 0,Y 526.047,Z 239.199,A -85,B 0,C 180,E1 22751.954,E2 22751.954} C_VEL
LIN {X 0,Y 525.922,Z 239.086,A -85,B 0,C 180,E1 22751.882,E2 22751.882} C_VEL
LIN {X 0,Y 524.728,Z 239.082,A -85,B 0,C 180,E1 22751.244,E2 22751.244} C_VEL
LIN {X 0,Y 521.116,Z 241.934,A -85,B 0,C 180,E1 22749.664,E2 22749.664} C_VEL
LIN {X 0,Y 520.4,Z 241.874,A -85,B 0,C 180,E1 22749.342,E2 22749.342} C_VEL
LIN {X 0,Y 517.093,Z 239.465,A -85,B 0,C 180,E1 22747.731,E2 22747.731} C_VEL
LIN {X 0,Y 514.463,Z 235.894,A -85,B 0,C 180,E1 22746.432,E2 22746.432} C_VEL
LIN {X 0,Y 513.826,Z 235.076,A -85,B 0,C 180,E1 22746.127,E2 22746.127} C_VEL
LIN {X 0,Y 510.249,Z 232.687,A -85,B 0,C 180,E1 22744.59,E2 22744.59} C_VEL
LIN {X 0,Y 507.59,Z 229.111,A -85,B 0,C 180,E1 22743.422,E2 22743.422} C_VEL
LIN {X 0,Y 506.839,Z 228.125,A -85,B 0,C 180,E1 22743.089,E2 22743.089} C_VEL
LIN {X 0,Y 503.527,Z 225.815,A -85,B 0,C 180,E1 22741.8,E2 22741.8} C_VEL
LIN {X 0,Y 500.752,Z 222.114,A -85,B 0,C 180,E1 22740.683,E2 22740.683} C_VEL
LIN {X 0,Y 500.077,Z 221.222,A -85,B 0,C 180,E1 22740.409,E2 22740.409} C_VEL
LIN {X 0,Y 496.637,Z 218.826,A -85,B 0,C 180,E1 22739.169,E2 22739.169} C_VEL
LIN {X 0,Y 494.31,Z 215.422,A -85,B 0,C 180,E1 22738.274,E2 22738.274} C_VEL
LIN {X 0,Y 493.728,Z 214.505,A -85,B 0,C 180,E1 22738.055,E2 22738.055} C_VEL
LIN {X 0,Y 490.418,Z 212.365,A -85,B 0,C 180,E1 22736.927,E2 22736.927} C_VEL
LIN {X 0,Y 488.273,Z 209.082,A -85,B 0,C 180,E1 22736.139,E2 22736.139} C_VEL
LIN {X 0,Y 487.499,Z 207.833,A -85,B 0,C 180,E1 22735.843,E2 22735.843} C_VEL
LIN {X 0,Y 484.242,Z 205.771,A -85,B 0,C 180,E1 22734.808,E2 22734.808} C_VEL
LIN {X 0,Y 482.484,Z 203.038,A -85,B 0,C 180,E1 22734.176,E2 22734.176} C_VEL
LIN {X 0,Y 482.03,Z 201.504,A -85,B 0,C 180,E1 22733.796,E2 22733.796} C_VEL
LIN {X 0,Y 482.019,Z 201.125,A -85,B 0,C 180,E1 22732.412,E2 22732.412} C_VEL
LIN {X 0,Y 481.976,Z 201.13,A -85,B 0,C 180,E1 22729.038,E2 22729.038} C_VEL
LIN {X 0,Y 481.962,Z 201.135,A -85,B 0,C 180,E1 22725.483,E2 22725.483} C_VEL
LIN {X 0,Y 481.972,Z 201.133,A -85,B 0,C 180,E1 22721.914,E2 22721.914} C_VEL
LIN {X 0,Y 482.018,Z 201.129,A -85,B 0,C 180,E1 22718.486,E2 22718.486} C_VEL
LIN {X 0,Y 481.985,Z 201.067,A -85,B 0,C 180,E1 22714.93,E2 22714.93} C_VEL
LIN {X 0,Y 481.963,Z 201.133,A -85,B 0,C 180,E1 22711.51,E2 22711.51} C_VEL
LIN {X 0,Y 481.955,Z 201.055,A -85,B 0,C 180,E1 22707.827,E2 22707.827} C_VEL
LIN {X 0,Y 481.991,Z 201.125,A -85,B 0,C 180,E1 22704.383,E2 22704.383} C_VEL
LIN {X 0,Y 482.012,Z 201.109,A -85,B 0,C 180,E1 22700.904,E2 22700.904} C_VEL
LIN {X 0,Y 481.974,Z 201.112,A -85,B 0,C 180,E1 22697.382,E2 22697.382} C_VEL
LIN {X 0,Y 481.96,Z 201.127,A -85,B 0,C 180,E1 22693.881,E2 22693.881} C_VEL
LIN {X 0,Y 481.98,Z 201.129,A -85,B 0,C 180,E1 22690.398,E2 22690.398} C_VEL
LIN {X 0,Y 482.024,Z 201.103,A -85,B 0,C 180,E1 22686.91,E2 22686.91} C_VEL
LIN {X 0,Y 481.986,Z 201.116,A -85,B 0,C 180,E1 22683.33,E2 22683.33} C_VEL
LIN {X 0,Y 481.961,Z 201.13,A -85,B 0,C 180,E1 22679.881,E2 22679.881} C_VEL
LIN {X 0,Y 481.96,Z 201.115,A -85,B 0,C 180,E1 22676.193,E2 22676.193} C_VEL
LIN {X 0,Y 481.987,Z 201.105,A -85,B 0,C 180,E1 22672.73,E2 22672.73} C_VEL
LIN {X 0,Y 482.01,Z 201.126,A -85,B 0,C 180,E1 22669.24,E2 22669.24} C_VEL
LIN {X 0,Y 481.976,Z 201.123,A -85,B 0,C 180,E1 22665.707,E2 22665.707} C_VEL
LIN {X 0,Y 481.961,Z 201.111,A -85,B 0,C 180,E1 22662.199,E2 22662.199} C_VEL
LIN {X 0,Y 481.971,Z 201.116,A -85,B 0,C 180,E1 22658.648,E2 22658.648} C_VEL
LIN {X 0,Y 482.017,Z 201.123,A -85,B 0,C 180,E1 22655.227,E2 22655.227} C_VEL
LIN {X 0,Y 481.99,Z 201.055,A -85,B 0,C 180,E1 22651.636,E2 22651.636} C_VEL
LIN {X 0,Y 481.967,Z 201.131,A -85,B 0,C 180,E1 22648.2,E2 22648.2} C_VEL
LIN {X 0,Y 481.961,Z 201.093,A -85,B 0,C 180,E1 22644.609,E2 22644.609} C_VEL
LIN {X 0,Y 482.002,Z 201.106,A -85,B 0,C 180,E1 22641.209,E2 22641.209} C_VEL
LIN {X 0,Y 481.999,Z 201.131,A -85,B 0,C 180,E1 22637.768,E2 22637.768} C_VEL
LIN {X 0,Y 482.003,Z 201.283,A -85,B 0,C 180,E1 22635.015,E2 22635.015} C_VEL
LIN {X 0,Y 487.68,Z 217.199,A -85,B 0,C 180,E1 22632.08,E2 22632.08} C_VEL
LIN {X 0,Y 488.601,Z 219.595,A -85,B 0,C 180,E1 22631.739,E2 22631.739} C_VEL
LIN {X 0,Y 499.285,Z 238.032,A -85,B 0,C 180,E1 22630.314,E2 22630.314} C_VEL
LIN {X 0,Y 510.997,Z 259.891,A -85,B 0,C 180,E1 22628.828,E2 22628.828} C_VEL
LIN {X 0,Y 517.732,Z 273.898,A -85,B 0,C 180,E1 22627.992,E2 22627.992} C_VEL
LIN {X 0,Y 518.476,Z 279.076,A -85,B 0,C 180,E1 22627.84,E2 22627.84} C_VEL
LIN {X 0,Y 511.366,Z 522.537,A -85,B 0,C 180,E1 22624.27,E2 22624.27} C_VEL
LIN {X 0,Y 510.301,Z 540.517,A -85,B 0,C 180,E1 22623.896,E2 22623.896} C_VEL
LIN {X 0,Y 508.696,Z 560.301,A -85,B 0,C 180,E1 22623.337,E2 22623.337} C_VEL
LIN {X 0,Y 506.366,Z 582.745,A -85,B 0,C 180,E1 22622.481,E2 22622.481} C_VEL
LIN {X 0,Y 504.188,Z 600.427,A -85,B 0,C 180,E1 22621.633,E2 22621.633} C_VEL
LIN {X 0,Y 502.005,Z 616.439,A -85,B 0,C 180,E1 22620.719,E2 22620.719} C_VEL
LIN {X 0,Y 499.681,Z 632.003,A -85,B 0,C 180,E1 22619.683,E2 22619.683} C_VEL
LIN {X 0,Y 497.414,Z 646.375,A -85,B 0,C 180,E1 22618.578,E2 22618.578} C_VEL
LIN {X 0,Y 495.084,Z 660.385,A -85,B 0,C 180,E1 22617.349,E2 22617.349} C_VEL
LIN {X 0,Y 492.742,Z 674.074,A -85,B 0,C 180,E1 22615.979,E2 22615.979} C_VEL
LIN {X 0,Y 490.236,Z 688.504,A -85,B 0,C 180,E1 22614.327,E2 22614.327} C_VEL
LIN {X 0,Y 487.481,Z 704.531,A -85,B 0,C 180,E1 22612.17,E2 22612.17} C_VEL
LIN {X 0,Y 485.446,Z 716.702,A -85,B 0,C 180,E1 22610.242,E2 22610.242} C_VEL
LIN {X 0,Y 483.901,Z 726.677,A -85,B 0,C 180,E1 22608.427,E2 22608.427} C_VEL
LIN {X 0,Y 482.665,Z 735.395,A -85,B 0,C 180,E1 22606.609,E2 22606.609} C_VEL
LIN {X 0,Y 481.653,Z 743.448,A -85,B 0,C 180,E1 22604.669,E2 22604.669} C_VEL
LIN {X 0,Y 480.925,Z 750.32,A -85,B 0,C 180,E1 22602.73,E2 22602.73} C_VEL
LIN {X 0,Y 480.419,Z 756.43,A -85,B 0,C 180,E1 22600.673,E2 22600.673} C_VEL
LIN {X 0,Y 480.087,Z 762.19,A -85,B 0,C 180,E1 22598.261,E2 22598.261} C_VEL
LIN {X 0,Y 479.943,Z 766.835,A -85,B 0,C 180,E1 22595.499,E2 22595.499} C_VEL
LIN {X 0,Y 479.925,Z 769.155,A -85,B 0,C 180,E1 22593.344,E2 22593.344} C_VEL
LIN {X 0,Y 479.931,Z 770.309,A -85,B 0,C 180,E1 22591.313,E2 22591.313} C_VEL
LIN {X 0,Y 479.937,Z 770.456,A -85,B 0,C 180,E1 22589.284,E2 22589.284} C_VEL
LIN {X 0,Y 479.927,Z 769.596,A -85,B 0,C 180,E1 22587.254,E2 22587.254} C_VEL
LIN {X 0,Y 479.927,Z 767.722,A -85,B 0,C 180,E1 22585.22,E2 22585.22} C_VEL
LIN {X 0,Y 479.98,Z 764.813,A -85,B 0,C 180,E1 22583.181,E2 22583.181} C_VEL
LIN {X 0,Y 480.135,Z 760.841,A -85,B 0,C 180,E1 22581.136,E2 22581.136} C_VEL
LIN {X 0,Y 480.467,Z 755.763,A -85,B 0,C 180,E1 22579.085,E2 22579.085} C_VEL
LIN {X 0,Y 480.963,Z 749.921,A -85,B 0,C 180,E1 22577.149,E2 22577.149} C_VEL
LIN {X 0,Y 481.707,Z 742.979,A -85,B 0,C 180,E1 22575.21,E2 22575.21} C_VEL
LIN {X 0,Y 482.739,Z 734.854,A -85,B 0,C 180,E1 22573.27,E2 22573.27} C_VEL
LIN {X 0,Y 484.188,Z 724.82,A -85,B 0,C 180,E1 22571.209,E2 22571.209} C_VEL
LIN {X 0,Y 486.417,Z 710.864,A -85,B 0,C 180,E1 22568.793,E2 22568.793} C_VEL
LIN {X 0,Y 488.483,Z 698.574,A -85,B 0,C 180,E1 22566.989,E2 22566.989} C_VEL
LIN {X 0,Y 490.721,Z 685.68,A -85,B 0,C 180,E1 22565.336,E2 22565.336} C_VEL
LIN {X 0,Y 492.953,Z 672.832,A -85,B 0,C 180,E1 22563.89,E2 22563.89} C_VEL
LIN {X 0,Y 495.297,Z 659.124,A -85,B 0,C 180,E1 22562.534,E2 22562.534} C_VEL
LIN {X 0,Y 497.755,Z 644.27,A -85,B 0,C 180,E1 22561.249,E2 22561.249} C_VEL
LIN {X 0,Y 500.779,Z 625.199,A -85,B 0,C 180,E1 22559.833,E2 22559.833} C_VEL
LIN {X 0,Y 503.555,Z 605.352,A -85,B 0,C 180,E1 22558.632,E2 22558.632} C_VEL
LIN {X 0,Y 505.635,Z 588.966,A -85,B 0,C 180,E1 22557.801,E2 22557.801} C_VEL
LIN {X 0,Y 507.49,Z 572.324,A -85,B 0,C 180,E1 22557.096,E2 22557.096} C_VEL
LIN {X 0,Y 509.131,Z 555.097,A -85,B 0,C 180,E1 22556.504,E2 22556.504} C_VEL
LIN {X 0,Y 510.47,Z 538.009,A -85,B 0,C 180,E1 22556.045,E2 22556.045} C_VEL
LIN {X 0,Y 511.465,Z 520.277,A -85,B 0,C 180,E1 22555.691,E2 22555.691} C_VEL
LIN {X 0,Y 518.475,Z 277.756,A -85,B 0,C 180,E1 22552.138,E2 22552.138} C_VEL
LIN {X 0,Y 517.201,Z 272.442,A -85,B 0,C 180,E1 22551.937,E2 22551.937} C_VEL
LIN {X 0,Y 505.164,Z 248.743,A -85,B 0,C 180,E1 22550.44,E2 22550.44} C_VEL
LIN {X 0,Y 494.205,Z 229.043,A -85,B 0,C 180,E1 22549.019,E2 22549.019} C_VEL
LIN {X 0,Y 488.178,Z 218.628,A -85,B 0,C 180,E1 22548.159,E2 22548.159} C_VEL
LIN {X 0,Y 483.029,Z 204.251,A -85,B 0,C 180,E1 22545.575,E2 22545.575} C_VEL
LIN {X 0,Y 481.994,Z 201.187,A -85,B 0,C 180,E1 22544.939,E2 22544.939} C_VEL
LIN {X 0,Y 481.963,Z 201.116,A -85,B 0,C 180,E1 22541.438,E2 22541.438} C_VEL
LIN {X 0,Y 481.966,Z 201.134,A -85,B 0,C 180,E1 22537.785,E2 22537.785} C_VEL
LIN {X 0,Y 481.996,Z 201.09,A -85,B 0,C 180,E1 22534.351,E2 22534.351} C_VEL
LIN {X 0,Y 482.009,Z 201.108,A -85,B 0,C 180,E1 22530.823,E2 22530.823} C_VEL
LIN {X 0,Y 481.963,Z 201.065,A -85,B 0,C 180,E1 22527.4,E2 22527.4} C_VEL
LIN {X 0,Y 481.962,Z 201.131,A -85,B 0,C 180,E1 22523.825,E2 22523.825} C_VEL
LIN {X 0,Y 481.987,Z 201.128,A -85,B 0,C 180,E1 22520.355,E2 22520.355} C_VEL
LIN {X 0,Y 482.015,Z 201.105,A -85,B 0,C 180,E1 22516.883,E2 22516.883} C_VEL
LIN {X 0,Y 481.971,Z 201.11,A -85,B 0,C 180,E1 22513.436,E2 22513.436} C_VEL
LIN {X 0,Y 481.961,Z 201.127,A -85,B 0,C 180,E1 22509.916,E2 22509.916} C_VEL
LIN {X 0,Y 481.978,Z 201.124,A -85,B 0,C 180,E1 22506.432,E2 22506.432} C_VEL
LIN {X 0,Y 482.009,Z 201.105,A -85,B 0,C 180,E1 22502.973,E2 22502.973} C_VEL
LIN {X 0,Y 481.975,Z 201.129,A -85,B 0,C 180,E1 22499.525,E2 22499.525} C_VEL
LIN {X 0,Y 481.959,Z 201.129,A -85,B 0,C 180,E1 22496.074,E2 22496.074} C_VEL
LIN {X 0,Y 481.972,Z 201.11,A -85,B 0,C 180,E1 22492.53,E2 22492.53} C_VEL
LIN {X 0,Y 482.013,Z 201.116,A -85,B 0,C 180,E1 22489.119,E2 22489.119} C_VEL
LIN {X 0,Y 481.982,Z 201.129,A -85,B 0,C 180,E1 22485.585,E2 22485.585} C_VEL
LIN {X 0,Y 481.962,Z 201.121,A -85,B 0,C 180,E1 22482.119,E2 22482.119} C_VEL
LIN {X 0,Y 481.968,Z 201.112,A -85,B 0,C 180,E1 22478.584,E2 22478.584} C_VEL
LIN {X 0,Y 482.014,Z 201.114,A -85,B 0,C 180,E1 22475.227,E2 22475.227} C_VEL
LIN {X 0,Y 481.988,Z 201.055,A -85,B 0,C 180,E1 22471.636,E2 22471.636} C_VEL
LIN {X 0,Y 481.964,Z 201.133,A -85,B 0,C 180,E1 22468.2,E2 22468.2} C_VEL
LIN {X 0,Y 481.956,Z 201.071,A -85,B 0,C 180,E1 22464.61,E2 22464.61} C_VEL
LIN {X 0,Y 482.006,Z 201.129,A -85,B 0,C 180,E1 22461.209,E2 22461.209} C_VEL
LIN {X 0,Y 481.995,Z 201.131,A -85,B 0,C 180,E1 22457.768,E2 22457.768} C_VEL
LIN {X 0,Y 481.965,Z 201.135,A -85,B 0,C 180,E1 22454.296,E2 22454.296} C_VEL
LIN {X 0,Y 481.964,Z 201.131,A -85,B 0,C 180,E1 22450.643,E2 22450.643} C_VEL
LIN {X 0,Y 481.988,Z 201.132,A -85,B 0,C 180,E1 22447.192,E2 22447.192} C_VEL
LIN {X 0,Y 482.029,Z 201.501,A -85,B 0,C 180,E1 22446.204,E2 22446.204} C_VEL
LIN {X 0,Y 482.527,Z 203.143,A -85,B 0,C 180,E1 22445.805,E2 22445.805} C_VEL
LIN {X 0,Y 484.333,Z 205.864,A -85,B 0,C 180,E1 22445.161,E2 22445.161} C_VEL
LIN {X 0,Y 487.999,Z 208.419,A -85,B 0,C 180,E1 22443.975,E2 22443.975} C_VEL
LIN {X 0,Y 489.875,Z 211.762,A -85,B 0,C 180,E1 22443.261,E2 22443.261} C_VEL
LIN {X 0,Y 492.843,Z 214.096,A -85,B 0,C 180,E1 22442.243,E2 22442.243} C_VEL
LIN {X 0,Y 494.064,Z 214.91,A -85,B 0,C 180,E1 22441.823,E2 22441.823} C_VEL
LIN {X 0,Y 496.341,Z 218.496,A -85,B 0,C 180,E1 22440.942,E2 22440.942} C_VEL
LIN {X 0,Y 499.311,Z 220.814,A -85,B 0,C 180,E1 22439.876,E2 22439.876} C_VEL
LIN {X 0,Y 500.56,Z 221.743,A -85,B 0,C 180,E1 22439.398,E2 22439.398} C_VEL
LIN {X 0,Y 503.216,Z 225.475,A -85,B 0,C 180,E1 22438.328,E2 22438.328} C_VEL
LIN {X 0,Y 506.44,Z 227.929,A -85,B 0,C 180,E1 22437.072,E2 22437.072} C_VEL
LIN {X 0,Y 507.407,Z 228.768,A -85,B 0,C 180,E1 22436.663,E2 22436.663} C_VEL
LIN {X 0,Y 510.095,Z 232.521,A -85,B 0,C 180,E1 22435.481,E2 22435.481} C_VEL
LIN {X 0,Y 513.518,Z 234.922,A -85,B 0,C 180,E1 22434.01,E2 22434.01} C_VEL
LIN {X 0,Y 514.396,Z 235.773,A -85,B 0,C 180,E1 22433.601,E2 22433.601} C_VEL
LIN {X 0,Y 516.958,Z 239.326,A -85,B 0,C 180,E1 22432.335,E2 22432.335} C_VEL
LIN {X 0,Y 520.034,Z 241.693,A -85,B 0,C 180,E1 22430.834,E2 22430.834} C_VEL
LIN {X 0,Y 521.495,Z 242.522,A -85,B 0,C 180,E1 22430.128,E2 22430.128} C_VEL
LIN {X 0,Y 524.189,Z 246.375,A -85,B 0,C 180,E1 22428.553,E2 22428.553} C_VEL
LIN {X 0,Y 527.271,Z 248.736,A -85,B 0,C 180,E1 22426.732,E2 22426.732} C_VEL
LIN {X 0,Y 529.141,Z 249.841,A -85,B 0,C 180,E1 22425.563,E2 22425.563} C_VEL
LIN {X 0,Y 531.128,Z 253.007,A -85,B 0,C 180,E1 22424.053,E2 22424.053} C_VEL
LIN {X 0,Y 533.761,Z 255.268,A -85,B 0,C 180,E1 22422,E2 22422} C_VEL
LIN {X 0,Y 536.533,Z 256.701,A -85,B 0,C 180,E1 22419.438,E2 22419.438} C_VEL
LIN {X 0,Y 537.666,Z 258.395,A -85,B 0,C 180,E1 22418.016,E2 22418.016} C_VEL
LIN {X 0,Y 539.124,Z 260.618,A -85,B 0,C 180,E1 22415.64,E2 22415.64} C_VEL
LIN {X 0,Y 540.208,Z 261.693,A -85,B 0,C 180,E1 22413.077,E2 22413.077} C_VEL
LIN {X 0,Y 540.652,Z 262.021,A -85,B 0,C 180,E1 22410.53,E2 22410.53} C_VEL
LIN {X 0,Y 540.474,Z 261.842,A -85,B 0,C 180,E1 22407.986,E2 22407.986} C_VEL
LIN {X 0,Y 539.693,Z 261.186,A -85,B 0,C 180,E1 22405.538,E2 22405.538} C_VEL
LIN {X 0,Y 538.549,Z 259.74,A -85,B 0,C 180,E1 22403.284,E2 22403.284} C_VEL
LIN {X 0,Y 537.421,Z 257.889,A -85,B 0,C 180,E1 22401.657,E2 22401.657} C_VEL
LIN {X 0,Y 536.074,Z 256.428,A -85,B 0,C 180,E1 22400.121,E2 22400.121} C_VEL
LIN {X 0,Y 533.473,Z 255.081,A -85,B 0,C 180,E1 22397.774,E2 22397.774} C_VEL
LIN {X 0,Y 530.978,Z 252.828,A -85,B 0,C 180,E1 22395.832,E2 22395.832} C_VEL
LIN {X 0,Y 528.645,Z 249.318,A -85,B 0,C 180,E1 22394.085,E2 22394.085} C_VEL
LIN {X 0,Y 525.19,Z 247.336,A -85,B 0,C 180,E1 22392.038,E2 22392.038} C_VEL
LIN {X 0,Y 522.412,Z 244.135,A -85,B 0,C 180,E1 22390.433,E2 22390.433} C_VEL
LIN {X 0,Y 521.126,Z 242.171,A -85,B 0,C 180,E1 22389.681,E2 22389.681} C_VEL
LIN {X 0,Y 520.4,Z 241.874,A -85,B 0,C 180,E1 22389.342,E2 22389.342} C_VEL
LIN {X 0,Y 517.834,Z 241.778,A -85,B 0,C 180,E1 22388.156,E2 22388.156} C_VEL
LIN {X 0,Y 513.107,Z 242.816,A -85,B 0,C 180,E1 22386.2,E2 22386.2} C_VEL
LIN {X 0,Y 511.488,Z 242.368,A -85,B 0,C 180,E1 22385.548,E2 22385.548} C_VEL
LIN {X 0,Y 508.258,Z 239.809,A -85,B 0,C 180,E1 22384.171,E2 22384.171} C_VEL
LIN {X 0,Y 505.382,Z 235.887,A -85,B 0,C 180,E1 22382.914,E2 22382.914} C_VEL
LIN {X 0,Y 501.928,Z 233.396,A -85,B 0,C 180,E1 22381.573,E2 22381.573} C_VEL
LIN {X 0,Y 498.91,Z 229.415,A -85,B 0,C 180,E1 22380.371,E2 22380.371} C_VEL
LIN {X 0,Y 494.73,Z 226.125,A -85,B 0,C 180,E1 22378.847,E2 22378.847} C_VEL
LIN {X 0,Y 491.799,Z 222.077,A -85,B 0,C 180,E1 22377.756,E2 22377.756} C_VEL
LIN {X 0,Y 488.476,Z 219.725,A -85,B 0,C 180,E1 22376.633,E2 22376.633} C_VEL
LIN {X 0,Y 486.095,Z 216.057,A -85,B 0,C 180,E1 22375.751,E2 22375.751} C_VEL
LIN {X 0,Y 485.124,Z 215.224,A -85,B 0,C 180,E1 22375.438,E2 22375.438} C_VEL
LIN {X 0,Y 482,Z 212.793,A -85,B 0,C 180,E1 22374.409,E2 22374.409} C_VEL
LIN {X 0,Y 479.946,Z 209.517,A -85,B 0,C 180,E1 22373.706,E2 22373.706} C_VEL
LIN {X 0,Y 479.182,Z 208.668,A -85,B 0,C 180,E1 22373.453,E2 22373.453} C_VEL
LIN {X 0,Y 476.309,Z 206.739,A -85,B 0,C 180,E1 22372.565,E2 22372.565} C_VEL
LIN {X 0,Y 474.417,Z 203.749,A -85,B 0,C 180,E1 22371.915,E2 22371.915} C_VEL
LIN {X 0,Y 474.053,Z 202.342,A -85,B 0,C 180,E1 22371.493,E2 22371.493} C_VEL
LIN {X 0,Y 474.071,Z 202.116,A -85,B 0,C 180,E1 22368.3,E2 22368.3} C_VEL
LIN {X 0,Y 474.072,Z 202.118,A -85,B 0,C 180,E1 22364.616,E2 22364.616} C_VEL
LIN {X 0,Y 474.035,Z 202.122,A -85,B 0,C 180,E1 22361.156,E2 22361.156} C_VEL
LIN {X 0,Y 474.022,Z 202.113,A -85,B 0,C 180,E1 22357.714,E2 22357.714} C_VEL
LIN {X 0,Y 474.041,Z 202.062,A -85,B 0,C 180,E1 22354.236,E2 22354.236} C_VEL
LIN {X 0,Y 474.084,Z 202.103,A -85,B 0,C 180,E1 22350.639,E2 22350.639} C_VEL
LIN {X 0,Y 474.039,Z 202.043,A -85,B 0,C 180,E1 22347.104,E2 22347.104} C_VEL
LIN {X 0,Y 474.024,Z 202.121,A -85,B 0,C 180,E1 22343.627,E2 22343.627} C_VEL
LIN {X 0,Y 474.026,Z 202.118,A -85,B 0,C 180,E1 22339.981,E2 22339.981} C_VEL
LIN {X 0,Y 474.057,Z 202.097,A -85,B 0,C 180,E1 22336.544,E2 22336.544} C_VEL
LIN {X 0,Y 474.068,Z 202.096,A -85,B 0,C 180,E1 22333.017,E2 22333.017} C_VEL
LIN {X 0,Y 474.037,Z 202.118,A -85,B 0,C 180,E1 22329.47,E2 22329.47} C_VEL
LIN {X 0,Y 474.021,Z 202.114,A -85,B 0,C 180,E1 22325.933,E2 22325.933} C_VEL
LIN {X 0,Y 474.025,Z 202.095,A -85,B 0,C 180,E1 22322.297,E2 22322.297} C_VEL
LIN {X 0,Y 474.063,Z 202.109,A -85,B 0,C 180,E1 22318.791,E2 22318.791} C_VEL
LIN {X 0,Y 474.071,Z 202.109,A -85,B 0,C 180,E1 22315.16,E2 22315.16} C_VEL
LIN {X 0,Y 474.028,Z 202.092,A -85,B 0,C 180,E1 22311.753,E2 22311.753} C_VEL
LIN {X 0,Y 474.023,Z 202.108,A -85,B 0,C 180,E1 22308.193,E2 22308.193} C_VEL
LIN {X 0,Y 474.043,Z 202.119,A -85,B 0,C 180,E1 22304.712,E2 22304.712} C_VEL
LIN {X 0,Y 474.074,Z 202.104,A -85,B 0,C 180,E1 22301.174,E2 22301.174} C_VEL
LIN {X 0,Y 474.046,Z 202.099,A -85,B 0,C 180,E1 22297.687,E2 22297.687} C_VEL
LIN {X 0,Y 474.022,Z 202.096,A -85,B 0,C 180,E1 22294.234,E2 22294.234} C_VEL
LIN {X 0,Y 474.02,Z 202.058,A -85,B 0,C 180,E1 22290.561,E2 22290.561} C_VEL
LIN {X 0,Y 474.067,Z 202.108,A -85,B 0,C 180,E1 22287.176,E2 22287.176} C_VEL
LIN {X 0,Y 474.073,Z 202.094,A -85,B 0,C 180,E1 22283.503,E2 22283.503} C_VEL
LIN {X 0,Y 474.027,Z 202.085,A -85,B 0,C 180,E1 22280.115,E2 22280.115} C_VEL
LIN {X 0,Y 474.023,Z 202.097,A -85,B 0,C 180,E1 22276.555,E2 22276.555} C_VEL
LIN {X 0,Y 474.115,Z 202.443,A -85,B 0,C 180,E1 22275.728,E2 22275.728} C_VEL
LIN {X 0,Y 479.798,Z 218.228,A -85,B 0,C 180,E1 22272.75,E2 22272.75} C_VEL
LIN {X 0,Y 484.884,Z 227.091,A -85,B 0,C 180,E1 22271.978,E2 22271.978} C_VEL
LIN {X 0,Y 493.879,Z 242.536,A -85,B 0,C 180,E1 22270.761,E2 22270.761} C_VEL
LIN {X 0,Y 505.58,Z 264.519,A -85,B 0,C 180,E1 22269.238,E2 22269.238} C_VEL
LIN {X 0,Y 511.794,Z 277.582,A -85,B 0,C 180,E1 22268.446,E2 22268.446} C_VEL
LIN {X 0,Y 512.093,Z 281.194,A -85,B 0,C 180,E1 22268.356,E2 22268.356} C_VEL
LIN {X 0,Y 504.76,Z 522.362,A -85,B 0,C 180,E1 22264.782,E2 22264.782} C_VEL
LIN {X 0,Y 503.663,Z 540.311,A -85,B 0,C 180,E1 22264.405,E2 22264.405} C_VEL
LIN {X 0,Y 502.001,Z 560.126,A -85,B 0,C 180,E1 22263.841,E2 22263.841} C_VEL
LIN {X 0,Y 499.589,Z 582.569,A -85,B 0,C 180,E1 22262.978,E2 22262.978} C_VEL
LIN {X 0,Y 497.33,Z 600.251,A -85,B 0,C 180,E1 22262.121,E2 22262.121} C_VEL
LIN {X 0,Y 495.021,Z 616.555,A -85,B 0,C 180,E1 22261.179,E2 22261.179} C_VEL
LIN {X 0,Y 492.694,Z 631.555,A -85,B 0,C 180,E1 22260.169,E2 22260.169} C_VEL
LIN {X 0,Y 490.291,Z 646.197,A -85,B 0,C 180,E1 22259.032,E2 22259.032} C_VEL
LIN {X 0,Y 487.865,Z 660.207,A -85,B 0,C 180,E1 22257.788,E2 22257.788} C_VEL
LIN {X 0,Y 485.442,Z 673.776,A -85,B 0,C 180,E1 22256.413,E2 22256.413} C_VEL
LIN {X 0,Y 482.809,Z 688.325,A -85,B 0,C 180,E1 22254.726,E2 22254.726} C_VEL
LIN {X 0,Y 479.916,Z 704.352,A -85,B 0,C 180,E1 22252.539,E2 22252.539} C_VEL
LIN {X 0,Y 477.78,Z 716.523,A -85,B 0,C 180,E1 22250.581,E2 22250.581} C_VEL
LIN {X 0,Y 476.135,Z 726.602,A -85,B 0,C 180,E1 22248.718,E2 22248.718} C_VEL
LIN {X 0,Y 474.844,Z 735.217,A -85,B 0,C 180,E1 22246.891,E2 22246.891} C_VEL
LIN {X 0,Y 473.77,Z 743.27,A -85,B 0,C 180,E1 22244.918,E2 22244.918} C_VEL
LIN {X 0,Y 472.996,Z 750.143,A -85,B 0,C 180,E1 22242.947,E2 22242.947} C_VEL
LIN {X 0,Y 472.457,Z 756.253,A -85,B 0,C 180,E1 22240.855,E2 22240.855} C_VEL
LIN {X 0,Y 472.089,Z 762.284,A -85,B 0,C 180,E1 22238.28,E2 22238.28} C_VEL
LIN {X 0,Y 471.947,Z 766.66,A -85,B 0,C 180,E1 22235.592,E2 22235.592} C_VEL
LIN {X 0,Y 471.926,Z 768.98,A -85,B 0,C 180,E1 22233.401,E2 22233.401} C_VEL
LIN {X 0,Y 471.933,Z 770.134,A -85,B 0,C 180,E1 22231.335,E2 22231.335} C_VEL
LIN {X 0,Y 471.938,Z 770.281,A -85,B 0,C 180,E1 22229.272,E2 22229.272} C_VEL
LIN {X 0,Y 471.928,Z 769.421,A -85,B 0,C 180,E1 22227.207,E2 22227.207} C_VEL
LIN {X 0,Y 471.926,Z 767.546,A -85,B 0,C 180,E1 22225.139,E2 22225.139} C_VEL
LIN {X 0,Y 471.985,Z 764.637,A -85,B 0,C 180,E1 22223.065,E2 22223.065} C_VEL
LIN {X 0,Y 472.153,Z 760.665,A -85,B 0,C 180,E1 22220.985,E2 22220.985} C_VEL
LIN {X 0,Y 472.506,Z 755.586,A -85,B 0,C 180,E1 22218.899,E2 22218.899} C_VEL
LIN {X 0,Y 473.037,Z 749.743,A -85,B 0,C 180,E1 22216.93,E2 22216.93} C_VEL
LIN {X 0,Y 473.827,Z 742.801,A -85,B 0,C 180,E1 22214.958,E2 22214.958} C_VEL
LIN {X 0,Y 474.923,Z 734.675,A -85,B 0,C 180,E1 22212.986,E2 22212.986} C_VEL
LIN {X 0,Y 476.454,Z 724.641,A -85,B 0,C 180,E1 22210.893,E2 22210.893} C_VEL
LIN {X 0,Y 478.798,Z 710.685,A -85,B 0,C 180,E1 22208.439,E2 22208.439} C_VEL
LIN {X 0,Y 480.972,Z 698.396,A -85,B 0,C 180,E1 22206.608,E2 22206.608} C_VEL
LIN {X 0,Y 483.202,Z 686.119,A -85,B 0,C 180,E1 22205.007,E2 22205.007} C_VEL
LIN {X 0,Y 485.542,Z 673.215,A -85,B 0,C 180,E1 22203.527,E2 22203.527} C_VEL
LIN {X 0,Y 487.975,Z 659.576,A -85,B 0,C 180,E1 22202.152,E2 22202.152} C_VEL
LIN {X 0,Y 490.41,Z 645.486,A -85,B 0,C 180,E1 22200.908,E2 22200.908} C_VEL
LIN {X 0,Y 492.911,Z 630.213,A -85,B 0,C 180,E1 22199.733,E2 22199.733} C_VEL
LIN {X 0,Y 495.603,Z 612.79,A -85,B 0,C 180,E1 22198.585,E2 22198.585} C_VEL
LIN {X 0,Y 498.537,Z 591.275,A -85,B 0,C 180,E1 22197.422,E2 22197.422} C_VEL
LIN {X 0,Y 500.674,Z 572.891,A -85,B 0,C 180,E1 22196.625,E2 22196.625} C_VEL
LIN {X 0,Y 502.404,Z 555.439,A -85,B 0,C 180,E1 22196.014,E2 22196.014} C_VEL
LIN {X 0,Y 503.804,Z 538.276,A -85,B 0,C 180,E1 22195.546,E2 22195.546} C_VEL
LIN {X 0,Y 504.839,Z 520.615,A -85,B 0,C 180,E1 22195.187,E2 22195.187} C_VEL
LIN {X 0,Y 512.109,Z 279.266,A -85,B 0,C 180,E1 22191.611,E2 22191.611} C_VEL
LIN {X 0,Y 511.143,Z 275.829,A -85,B 0,C 180,E1 22191.466,E2 22191.466} C_VEL
LIN {X 0,Y 499.624,Z 253.088,A -85,B 0,C 180,E1 22189.996,E2 22189.996} C_VEL
LIN {X 0,Y 489.004,Z 233.912,A -85,B 0,C 180,E1 22188.583,E2 22188.583} C_VEL
LIN {X 0,Y 479.852,Z 218.37,A -85,B 0,C 180,E1 22187.267,E2 22187.267} C_VEL
LIN {X 0,Y 474.811,Z 204.609,A -85,B 0,C 180,E1 22184.698,E2 22184.698} C_VEL
LIN {X 0,Y 474.071,Z 202.21,A -85,B 0,C 180,E1 22184.191,E2 22184.191} C_VEL
LIN {X 0,Y 474.08,Z 202.081,A -85,B 0,C 180,E1 22180.512,E2 22180.512} C_VEL
LIN {X 0,Y 474.051,Z 202.11,A -85,B 0,C 180,E1 22176.937,E2 22176.937} C_VEL
LIN {X 0,Y 474.026,Z 202.1,A -85,B 0,C 180,E1 22173.364,E2 22173.364} C_VEL
LIN {X 0,Y 474.021,Z 202.068,A -85,B 0,C 180,E1 22169.856,E2 22169.856} C_VEL
LIN {X 0,Y 474.055,Z 202.072,A -85,B 0,C 180,E1 22166.427,E2 22166.427} C_VEL
LIN {X 0,Y 474.079,Z 202.099,A -85,B 0,C 180,E1 22162.835,E2 22162.835} C_VEL
LIN {X 0,Y 474.037,Z 202.118,A -85,B 0,C 180,E1 22159.339,E2 22159.339} C_VEL
LIN {X 0,Y 474.023,Z 202.116,A -85,B 0,C 180,E1 22155.79,E2 22155.79} C_VEL
LIN {X 0,Y 474.034,Z 202.099,A -85,B 0,C 180,E1 22152.301,E2 22152.301} C_VEL
LIN {X 0,Y 474.067,Z 202.093,A -85,B 0,C 180,E1 22148.735,E2 22148.735} C_VEL
LIN {X 0,Y 474.06,Z 202.119,A -85,B 0,C 180,E1 22145.204,E2 22145.204} C_VEL
LIN {X 0,Y 474.027,Z 202.11,A -85,B 0,C 180,E1 22141.692,E2 22141.692} C_VEL
LIN {X 0,Y 474.019,Z 202.097,A -85,B 0,C 180,E1 22138.066,E2 22138.066} C_VEL
LIN {X 0,Y 474.037,Z 202.114,A -85,B 0,C 180,E1 22134.536,E2 22134.536} C_VEL
LIN {X 0,Y 474.076,Z 202.11,A -85,B 0,C 180,E1 22131.021,E2 22131.021} C_VEL
LIN {X 0,Y 474.064,Z 202.095,A -85,B 0,C 180,E1 22127.329,E2 22127.329} C_VEL
LIN {X 0,Y 474.024,Z 202.109,A -85,B 0,C 180,E1 22123.959,E2 22123.959} C_VEL
LIN {X 0,Y 474.025,Z 202.12,A -85,B 0,C 180,E1 22120.404,E2 22120.404} C_VEL
LIN {X 0,Y 474.052,Z 202.116,A -85,B 0,C 180,E1 22116.901,E2 22116.901} C_VEL
LIN {X 0,Y 474.07,Z 202.047,A -85,B 0,C 180,E1 22113.304,E2 22113.304} C_VEL
LIN {X 0,Y 474.036,Z 202.092,A -85,B 0,C 180,E1 22109.848,E2 22109.848} C_VEL
LIN {X 0,Y 474.019,Z 202.079,A -85,B 0,C 180,E1 22106.418,E2 22106.418} C_VEL
LIN {X 0,Y 474.032,Z 202.091,A -85,B 0,C 180,E1 22102.865,E2 22102.865} C_VEL
LIN {X 0,Y 474.086,Z 202.116,A -85,B 0,C 180,E1 22099.391,E2 22099.391} C_VEL
LIN {X 0,Y 474.063,Z 202.118,A -85,B 0,C 180,E1 22095.722,E2 22095.722} C_VEL
LIN {X 0,Y 474.029,Z 202.12,A -85,B 0,C 180,E1 22092.236,E2 22092.236} C_VEL
LIN {X 0,Y 474.031,Z 202.189,A -85,B 0,C 180,E1 22088.629,E2 22088.629} C_VEL
LIN {X 0,Y 474.318,Z 203.454,A -85,B 0,C 180,E1 22088.132,E2 22088.132} C_VEL
LIN {X 0,Y 476.035,Z 206.44,A -85,B 0,C 180,E1 22087.521,E2 22087.521} C_VEL
LIN {X 0,Y 478.787,Z 208.484,A -85,B 0,C 180,E1 22086.669,E2 22086.669} C_VEL
LIN {X 0,Y 479.899,Z 209.407,A -85,B 0,C 180,E1 22086.311,E2 22086.311} C_VEL
LIN {X 0,Y 481.875,Z 212.652,A -85,B 0,C 180,E1 22085.632,E2 22085.632} C_VEL
LIN {X 0,Y 484.887,Z 215.105,A -85,B 0,C 180,E1 22084.635,E2 22084.635} C_VEL
LIN {X 0,Y 486.036,Z 215.934,A -85,B 0,C 180,E1 22084.271,E2 22084.271} C_VEL
LIN {X 0,Y 488.337,Z 219.573,A -85,B 0,C 180,E1 22083.416,E2 22083.416} C_VEL
LIN {X 0,Y 491.516,Z 221.941,A -85,B 0,C 180,E1 22082.34,E2 22082.34} C_VEL
LIN {X 0,Y 492.295,Z 222.618,A -85,B 0,C 180,E1 22082.062,E2 22082.062} C_VEL
LIN {X 0,Y 494.949,Z 226.369,A -85,B 0,C 180,E1 22081.067,E2 22081.067} C_VEL
LIN {X 0,Y 498.394,Z 228.867,A -85,B 0,C 180,E1 22079.833,E2 22079.833} C_VEL
LIN {X 0,Y 502.138,Z 233.615,A -85,B 0,C 180,E1 22078.34,E2 22078.34} C_VEL
LIN {X 0,Y 505.882,Z 236.503,A -85,B 0,C 180,E1 22076.866,E2 22076.866} C_VEL
LIN {X 0,Y 508.835,Z 240.412,A -85,B 0,C 180,E1 22075.582,E2 22075.582} C_VEL
LIN {X 0,Y 512.611,Z 242.942,A -85,B 0,C 180,E1 22073.963,E2 22073.963} C_VEL
LIN {X 0,Y 515.563,Z 247.028,A -85,B 0,C 180,E1 22072.518,E2 22072.518} C_VEL
LIN {X 0,Y 518.971,Z 249.629,A -85,B 0,C 180,E1 22070.862,E2 22070.862} C_VEL
LIN {X 0,Y 520.259,Z 250.49,A -85,B 0,C 180,E1 22070.237,E2 22070.237} C_VEL
LIN {X 0,Y 523.165,Z 254.411,A -85,B 0,C 180,E1 22068.563,E2 22068.563} C_VEL
LIN {X 0,Y 526.389,Z 256.748,A -85,B 0,C 180,E1 22066.666,E2 22066.666} C_VEL
LIN {X 0,Y 527.93,Z 257.643,A -85,B 0,C 180,E1 22065.712,E2 22065.712} C_VEL
LIN {X 0,Y 529.944,Z 260.809,A -85,B 0,C 180,E1 22064.197,E2 22064.197} C_VEL
LIN {X 0,Y 532.606,Z 263.115,A -85,B 0,C 180,E1 22062.136,E2 22062.136} C_VEL
LIN {X 0,Y 535.424,Z 264.565,A -85,B 0,C 180,E1 22059.566,E2 22059.566} C_VEL
LIN {X 0,Y 536.596,Z 266.238,A -85,B 0,C 180,E1 22058.14,E2 22058.14} C_VEL
LIN {X 0,Y 538.071,Z 268.496,A -85,B 0,C 180,E1 22055.758,E2 22055.758} C_VEL
LIN {X 0,Y 539.193,Z 269.599,A -85,B 0,C 180,E1 22053.189,E2 22053.189} C_VEL
LIN {X 0,Y 539.668,Z 269.959,A -85,B 0,C 180,E1 22050.637,E2 22050.637} C_VEL
LIN {X 0,Y 539.499,Z 269.784,A -85,B 0,C 180,E1 22047.982,E2 22047.982} C_VEL
LIN {X 0,Y 538.713,Z 269.129,A -85,B 0,C 180,E1 22045.53,E2 22045.53} C_VEL
LIN {X 0,Y 537.561,Z 267.689,A -85,B 0,C 180,E1 22043.271,E2 22043.271} C_VEL
LIN {X 0,Y 536.331,Z 265.728,A -85,B 0,C 180,E1 22041.532,E2 22041.532} C_VEL
LIN {X 0,Y 535.008,Z 264.333,A -85,B 0,C 180,E1 22040.04,E2 22040.04} C_VEL
LIN {X 0,Y 532.296,Z 262.924,A -85,B 0,C 180,E1 22037.633,E2 22037.633} C_VEL
LIN {X 0,Y 529.796,Z 260.629,A -85,B 0,C 180,E1 22035.688,E2 22035.688} C_VEL
LIN {X 0,Y 527.469,Z 257.185,A -85,B 0,C 180,E1 22033.965,E2 22033.965} C_VEL
LIN {X 0,Y 524.12,Z 255.283,A -85,B 0,C 180,E1 22032,E2 22032} C_VEL
LIN {X 0,Y 521.264,Z 252.129,A -85,B 0,C 180,E1 22030.363,E2 22030.363} C_VEL
LIN {X 0,Y 519.745,Z 249.976,A -85,B 0,C 180,E1 22029.508,E2 22029.508} C_VEL
LIN {X 0,Y 516.214,Z 247.672,A -85,B 0,C 180,E1 22027.801,E2 22027.801} C_VEL
LIN {X 0,Y 513.351,Z 244.177,A -85,B 0,C 180,E1 22026.409,E2 22026.409} C_VEL
LIN {X 0,Y 512.38,Z 242.827,A -85,B 0,C 180,E1 22025.933,E2 22025.933} C_VEL
LIN {X 0,Y 511.488,Z 242.368,A -85,B 0,C 180,E1 22025.548,E2 22025.548} C_VEL
LIN {X 0,Y 509.755,Z 242.639,A -85,B 0,C 180,E1 22024.891,E2 22024.891} C_VEL
LIN {X 0,Y 506.058,Z 245.136,A -85,B 0,C 180,E1 22023.604,E2 22023.604} C_VEL
LIN {X 0,Y 504.615,Z 244.619,A -85,B 0,C 180,E1 22023.046,E2 22023.046} C_VEL
LIN {X 0,Y 504.444,Z 244.368,A -85,B 0,C 180,E1 22022.97,E2 22022.97} C_VEL
LIN {X 0,Y 503.407,Z 243.4,A -85,B 0,C 180,E1 22022.565,E2 22022.565} C_VEL
LIN {X 0,Y 499.847,Z 240.535,A -85,B 0,C 180,E1 22021.184,E2 22021.184} C_VEL
LIN {X 0,Y 496.636,Z 236.488,A -85,B 0,C 180,E1 22019.917,E2 22019.917} C_VEL
LIN {X 0,Y 493.051,Z 233.71,A -85,B 0,C 180,E1 22018.625,E2 22018.625} C_VEL
LIN {X 0,Y 490.191,Z 229.786,A -85,B 0,C 180,E1 22017.562,E2 22017.562} C_VEL
LIN {X 0,Y 486.547,Z 227.081,A -85,B 0,C 180,E1 22016.337,E2 22016.337} C_VEL
LIN {X 0,Y 483.559,Z 222.966,A -85,B 0,C 180,E1 22015.28,E2 22015.28} C_VEL
LIN {X 0,Y 480.118,Z 220.292,A -85,B 0,C 180,E1 22014.162,E2 22014.162} C_VEL
LIN {X 0,Y 477.729,Z 216.622,A -85,B 0,C 180,E1 22013.336,E2 22013.336} C_VEL
LIN {X 0,Y 474.104,Z 213.903,A -85,B 0,C 180,E1 22012.219,E2 22012.219} C_VEL
LIN {X 0,Y 471.886,Z 210.356,A -85,B 0,C 180,E1 22011.46,E2 22011.46} C_VEL
LIN {X 0,Y 470.076,Z 209.068,A -85,B 0,C 180,E1 22010.931,E2 22010.931} C_VEL
LIN {X 0,Y 467.317,Z 206.439,A -85,B 0,C 180,E1 22010.074,E2 22010.074} C_VEL
LIN {X 0,Y 466.2,Z 203.775,A -85,B 0,C 180,E1 22009.587,E2 22009.587} C_VEL
LIN {X 0,Y 466.096,Z 203.138,A -85,B 0,C 180,E1 22009.14,E2 22009.14} C_VEL
LIN {X 0,Y 466.085,Z 203.113,A -85,B 0,C 180,E1 22005.593,E2 22005.593} C_VEL
LIN {X 0,Y 466.101,Z 203.111,A -85,B 0,C 180,E1 22002.014,E2 22002.014} C_VEL
LIN {X 0,Y 466.137,Z 203.107,A -85,B 0,C 180,E1 21998.467,E2 21998.467} C_VEL
LIN {X 0,Y 466.117,Z 203.041,A -85,B 0,C 180,E1 21994.767,E2 21994.767} C_VEL
LIN {X 0,Y 466.095,Z 203.112,A -85,B 0,C 180,E1 21991.275,E2 21991.275} C_VEL
LIN {X 0,Y 466.077,Z 203.029,A -85,B 0,C 180,E1 21987.745,E2 21987.745} C_VEL
LIN {X 0,Y 466.098,Z 203.109,A -85,B 0,C 180,E1 21984.189,E2 21984.189} C_VEL
LIN {X 0,Y 466.138,Z 203.087,A -85,B 0,C 180,E1 21980.728,E2 21980.728} C_VEL
LIN {X 0,Y 466.117,Z 203.084,A -85,B 0,C 180,E1 21977.091,E2 21977.091} C_VEL
LIN {X 0,Y 466.085,Z 203.102,A -85,B 0,C 180,E1 21973.65,E2 21973.65} C_VEL
LIN {X 0,Y 466.085,Z 203.108,A -85,B 0,C 180,E1 21970.007,E2 21970.007} C_VEL
LIN {X 0,Y 466.104,Z 203.088,A -85,B 0,C 180,E1 21966.528,E2 21966.528} C_VEL
LIN {X 0,Y 466.13,Z 203.083,A -85,B 0,C 180,E1 21962.951,E2 21962.951} C_VEL
LIN {X 0,Y 466.11,Z 203.108,A -85,B 0,C 180,E1 21959.385,E2 21959.385} C_VEL
LIN {X 0,Y 466.088,Z 203.097,A -85,B 0,C 180,E1 21955.817,E2 21955.817} C_VEL
LIN {X 0,Y 466.082,Z 203.081,A -85,B 0,C 180,E1 21952.232,E2 21952.232} C_VEL
LIN {X 0,Y 466.109,Z 203.098,A -85,B 0,C 180,E1 21948.743,E2 21948.743} C_VEL
LIN {X 0,Y 466.142,Z 203.103,A -85,B 0,C 180,E1 21945.084,E2 21945.084} C_VEL
LIN {X 0,Y 466.13,Z 203.09,A -85,B 0,C 180,E1 21941.36,E2 21941.36} C_VEL
LIN {X 0,Y 466.096,Z 203.088,A -85,B 0,C 180,E1 21937.817,E2 21937.817} C_VEL
LIN {X 0,Y 466.084,Z 203.085,A -85,B 0,C 180,E1 21934.277,E2 21934.277} C_VEL
LIN {X 0,Y 466.087,Z 203.041,A -85,B 0,C 180,E1 21930.717,E2 21930.717} C_VEL
LIN {X 0,Y 466.131,Z 203.097,A -85,B 0,C 180,E1 21927.22,E2 21927.22} C_VEL
LIN {X 0,Y 466.13,Z 203.081,A -85,B 0,C 180,E1 21923.542,E2 21923.542} C_VEL
LIN {X 0,Y 466.089,Z 203.073,A -85,B 0,C 180,E1 21920.101,E2 21920.101} C_VEL
LIN {X 0,Y 466.111,Z 203.283,A -85,B 0,C 180,E1 21916.573,E2 21916.573} C_VEL
LIN {X 0,Y 471.489,Z 218.004,A -85,B 0,C 180,E1 21913.684,E2 21913.684} C_VEL
LIN {X 0,Y 482.365,Z 236.221,A -85,B 0,C 180,E1 21912.067,E2 21912.067} C_VEL
LIN {X 0,Y 493.868,Z 256.942,A -85,B 0,C 180,E1 21910.492,E2 21910.492} C_VEL
LIN {X 0,Y 505.154,Z 279.291,A -85,B 0,C 180,E1 21909.013,E2 21909.013} C_VEL
LIN {X 0,Y 505.815,Z 281.382,A -85,B 0,C 180,E1 21908.915,E2 21908.915} C_VEL
LIN {X 0,Y 498.195,Z 522.187,A -85,B 0,C 180,E1 21905.308,E2 21905.308} C_VEL
LIN {X 0,Y 497.054,Z 540.275,A -85,B 0,C 180,E1 21904.925,E2 21904.925} C_VEL
LIN {X 0,Y 495.286,Z 560.634,A -85,B 0,C 180,E1 21904.337,E2 21904.337} C_VEL
LIN {X 0,Y 492.851,Z 582.393,A -85,B 0,C 180,E1 21903.487,E2 21903.487} C_VEL
LIN {X 0,Y 490.512,Z 600.074,A -85,B 0,C 180,E1 21902.622,E2 21902.622} C_VEL
LIN {X 0,Y 488.122,Z 616.338,A -85,B 0,C 180,E1 21901.673,E2 21901.673} C_VEL
LIN {X 0,Y 485.791,Z 630.842,A -85,B 0,C 180,E1 21900.689,E2 21900.689} C_VEL
LIN {X 0,Y 483.351,Z 645.173,A -85,B 0,C 180,E1 21899.571,E2 21899.571} C_VEL
LIN {X 0,Y 480.791,Z 659.398,A -85,B 0,C 180,E1 21898.301,E2 21898.301} C_VEL
LIN {X 0,Y 478.252,Z 673.037,A -85,B 0,C 180,E1 21896.909,E2 21896.909} C_VEL
LIN {X 0,Y 475.696,Z 686.566,A -85,B 0,C 180,E1 21895.332,E2 21895.332} C_VEL
LIN {X 0,Y 472.842,Z 701.773,A -85,B 0,C 180,E1 21893.29,E2 21893.29} C_VEL
LIN {X 0,Y 470.264,Z 715.643,A -85,B 0,C 180,E1 21891.056,E2 21891.056} C_VEL
LIN {X 0,Y 468.52,Z 725.7,A -85,B 0,C 180,E1 21889.185,E2 21889.185} C_VEL
LIN {X 0,Y 467.116,Z 734.497,A -85,B 0,C 180,E1 21887.307,E2 21887.307} C_VEL
LIN {X 0,Y 465.956,Z 742.623,A -85,B 0,C 180,E1 21885.302,E2 21885.302} C_VEL
LIN {X 0,Y 465.117,Z 749.565,A -85,B 0,C 180,E1 21883.297,E2 21883.297} C_VEL
LIN {X 0,Y 464.522,Z 755.742,A -85,B 0,C 180,E1 21881.169,E2 21881.169} C_VEL
LIN {X 0,Y 464.158,Z 760.758,A -85,B 0,C 180,E1 21879.046,E2 21879.046} C_VEL
LIN {X 0,Y 463.977,Z 765.086,A -85,B 0,C 180,E1 21876.682,E2 21876.682} C_VEL
LIN {X 0,Y 463.932,Z 768.615,A -85,B 0,C 180,E1 21873.725,E2 21873.725} C_VEL
LIN {X 0,Y 463.935,Z 769.959,A -85,B 0,C 180,E1 21871.358,E2 21871.358} C_VEL
LIN {X 0,Y 463.94,Z 770.106,A -85,B 0,C 180,E1 21869.259,E2 21869.259} C_VEL
LIN {X 0,Y 463.928,Z 769.246,A -85,B 0,C 180,E1 21867.159,E2 21867.159} C_VEL
LIN {X 0,Y 463.927,Z 767.371,A -85,B 0,C 180,E1 21865.055,E2 21865.055} C_VEL
LIN {X 0,Y 463.992,Z 764.461,A -85,B 0,C 180,E1 21862.945,E2 21862.945} C_VEL
LIN {X 0,Y 464.175,Z 760.488,A -85,B 0,C 180,E1 21860.829,E2 21860.829} C_VEL
LIN {X 0,Y 464.55,Z 755.409,A -85,B 0,C 180,E1 21858.706,E2 21858.706} C_VEL
LIN {X 0,Y 465.118,Z 749.565,A -85,B 0,C 180,E1 21856.703,E2 21856.703} C_VEL
LIN {X 0,Y 465.957,Z 742.623,A -85,B 0,C 180,E1 21854.698,E2 21854.698} C_VEL
LIN {X 0,Y 467.122,Z 734.463,A -85,B 0,C 180,E1 21852.685,E2 21852.685} C_VEL
LIN {X 0,Y 468.768,Z 724.271,A -85,B 0,C 180,E1 21850.527,E2 21850.527} C_VEL
LIN {X 0,Y 471.283,Z 710.017,A -85,B 0,C 180,E1 21847.996,E2 21847.996} C_VEL
LIN {X 0,Y 473.648,Z 697.327,A -85,B 0,C 180,E1 21846.092,E2 21846.092} C_VEL
LIN {X 0,Y 475.956,Z 685.148,A -85,B 0,C 180,E1 21844.494,E2 21844.494} C_VEL
LIN {X 0,Y 478.461,Z 671.915,A -85,B 0,C 180,E1 21842.969,E2 21842.969} C_VEL
LIN {X 0,Y 481.105,Z 657.71,A -85,B 0,C 180,E1 21841.538,E2 21841.538} C_VEL
LIN {X 0,Y 484.237,Z 640.331,A -85,B 0,C 180,E1 21840.024,E2 21840.024} C_VEL
LIN {X 0,Y 487.464,Z 620.689,A -85,B 0,C 180,E1 21838.605,E2 21838.605} C_VEL
LIN {X 0,Y 489.914,Z 604.324,A -85,B 0,C 180,E1 21837.61,E2 21837.61} C_VEL
LIN {X 0,Y 492.213,Z 587.368,A -85,B 0,C 180,E1 21836.742,E2 21836.742} C_VEL
LIN {X 0,Y 494.125,Z 571.229,A -85,B 0,C 180,E1 21836.053,E2 21836.053} C_VEL
LIN {X 0,Y 495.879,Z 553.931,A -85,B 0,C 180,E1 21835.453,E2 21835.453} C_VEL
LIN {X 0,Y 497.325,Z 536.479,A -85,B 0,C 180,E1 21834.984,E2 21834.984} C_VEL
LIN {X 0,Y 498.429,Z 517.154,A -85,B 0,C 180,E1 21834.603,E2 21834.603} C_VEL
LIN {X 0,Y 505.784,Z 280.731,A -85,B 0,C 180,E1 21831.071,E2 21831.071} C_VEL
LIN {X 0,Y 494.614,Z 258.35,A -85,B 0,C 180,E1 21829.608,E2 21829.608} C_VEL
LIN {X 0,Y 483.825,Z 238.748,A -85,B 0,C 180,E1 21828.137,E2 21828.137} C_VEL
LIN {X 0,Y 473.936,Z 222.369,A -85,B 0,C 180,E1 21826.73,E2 21826.73} C_VEL
LIN {X 0,Y 471.399,Z 217.794,A -85,B 0,C 180,E1 21826.285,E2 21826.285} C_VEL
LIN {X 0,Y 466.918,Z 205.743,A -85,B 0,C 180,E1 21823.935,E2 21823.935} C_VEL
LIN {X 0,Y 466.099,Z 203.192,A -85,B 0,C 180,E1 21823.352,E2 21823.352} C_VEL
LIN {X 0,Y 466.081,Z 203.075,A -85,B 0,C 180,E1 21819.641,E2 21819.641} C_VEL
LIN {X 0,Y 466.104,Z 203.077,A -85,B 0,C 180,E1 21816.152,E2 21816.152} C_VEL
LIN {X 0,Y 466.138,Z 203.1,A -85,B 0,C 180,E1 21812.554,E2 21812.554} C_VEL
LIN {X 0,Y 466.107,Z 203.034,A -85,B 0,C 180,E1 21809.001,E2 21809.001} C_VEL
LIN {X 0,Y 466.091,Z 203.094,A -85,B 0,C 180,E1 21805.44,E2 21805.44} C_VEL
LIN {X 0,Y 466.082,Z 203.089,A -85,B 0,C 180,E1 21801.786,E2 21801.786} C_VEL
LIN {X 0,Y 466.1,Z 203.086,A -85,B 0,C 180,E1 21798.253,E2 21798.253} C_VEL
LIN {X 0,Y 466.132,Z 203.097,A -85,B 0,C 180,E1 21794.662,E2 21794.662} C_VEL
LIN {X 0,Y 466.129,Z 203.099,A -85,B 0,C 180,E1 21791.006,E2 21791.006} C_VEL
